LIN {X 0,Y 704.416,Z 634.552,A -85,B 0,C 180,E1 -3430.383,E2 -3430.383} C_VEL
LIN {X 0,Y 704.53,Z 624.148,A -85,B 0,C 180,E1 -3430.889,E2 -3430.889} C_VEL
LIN {X 0,Y 704.712,Z 613.331,A -85,B 0,C 180,E1 -3431.321,E2 -3431.321} C_VEL
LIN {X 0,Y 704.817,Z 602.117,A -85,B 0,C 180,E1 -3431.683,E2 -3431.683} C_VEL
LIN {X 0,Y 704.875,Z 590.492,A -85,B 0,C 180,E1 -3431.972,E2 -3431.972} C_VEL
LIN {X 0,Y 704.941,Z 578.231,A -85,B 0,C 180,E1 -3432.19,E2 -3432.19} C_VEL
LIN {X 0,Y 705.133,Z 516.872,A -85,B 0,C 180,E1 -3432.832,E2 -3432.832} C_VEL
LIN {X 0,Y 705.313,Z 446.172,A -85,B 0,C 180,E1 -3433.553,E2 -3433.553} C_VEL
LIN {X 0,Y 704.909,Z 442.652,A -85,B 0,C 180,E1 -3433.636,E2 -3433.636} C_VEL
LIN {X 0,Y 703.676,Z 438.808,A -85,B 0,C 180,E1 -3433.829,E2 -3433.829} C_VEL
LIN {X 0,Y 701.394,Z 434.303,A -85,B 0,C 180,E1 -3434.192,E2 -3434.192} C_VEL
LIN {X 0,Y 698.323,Z 427.937,A -85,B 0,C 180,E1 -3434.84,E2 -3434.84} C_VEL
LIN {X 0,Y 697.717,Z 423.757,A -85,B 0,C 180,E1 -3435.236,E2 -3435.236} C_VEL
LIN {X 0,Y 698.092,Z 392.579,A -85,B 0,C 180,E1 -3438.122,E2 -3438.122} C_VEL
LIN {X 0,Y 698.45,Z 360.795,A -85,B 0,C 180,E1 -3441.048,E2 -3441.048} C_VEL
LIN {X 0,Y 698.726,Z 332.913,A -85,B 0,C 180,E1 -3443.64,E2 -3443.64} C_VEL
LIN {X 0,Y 698.786,Z 319.402,A -85,B 0,C 180,E1 -3444.898,E2 -3444.898} C_VEL
LIN {X 0,Y 697.086,Z 311.216,A -85,B 0,C 180,E1 -3445.739,E2 -3445.739} C_VEL
LIN {X 0,Y 697.089,Z 311.207,A -85,B 0,C 180,E1 -3448.182,E2 -3448.182} C_VEL
LIN {X 0,Y 697.083,Z 311.208,A -85,B 0,C 180,E1 -3450.828,E2 -3450.828} C_VEL
LIN {X 0,Y 697.065,Z 311.215,A -85,B 0,C 180,E1 -3453.486,E2 -3453.486} C_VEL
LIN {X 0,Y 697.085,Z 311.208,A -85,B 0,C 180,E1 -3455.648,E2 -3455.648} C_VEL
LIN {X 0,Y 697.071,Z 311.207,A -85,B 0,C 180,E1 -3458.392,E2 -3458.392} C_VEL
LIN {X 0,Y 697.107,Z 311.212,A -85,B 0,C 180,E1 -3461.097,E2 -3461.097} C_VEL
LIN {X 0,Y 697.065,Z 311.208,A -85,B 0,C 180,E1 -3463.656,E2 -3463.656} C_VEL
LIN {X 0,Y 697.067,Z 311.207,A -85,B 0,C 180,E1 -3466.105,E2 -3466.105} C_VEL
LIN {X 0,Y 697.088,Z 311.21,A -85,B 0,C 180,E1 -3468.457,E2 -3468.457} C_VEL
LIN {X 0,Y 697.069,Z 311.218,A -85,B 0,C 180,E1 -3470.724,E2 -3470.724} C_VEL
LIN {X 0,Y 697.066,Z 311.207,A -85,B 0,C 180,E1 -3473.502,E2 -3473.502} C_VEL
LIN {X 0,Y 697.074,Z 311.207,A -85,B 0,C 180,E1 -3475.757,E2 -3475.757} C_VEL
LIN {X 0,Y 697.089,Z 311.214,A -85,B 0,C 180,E1 -3478.5,E2 -3478.5} C_VEL
LIN {X 0,Y 697.077,Z 311.206,A -85,B 0,C 180,E1 -3481.163,E2 -3481.163} C_VEL
LIN {X 0,Y 697.084,Z 311.205,A -85,B 0,C 180,E1 -3483.418,E2 -3483.418} C_VEL
LIN {X 0,Y 697.069,Z 311.218,A -85,B 0,C 180,E1 -3486.122,E2 -3486.122} C_VEL
LIN {X 0,Y 697.09,Z 311.205,A -85,B 0,C 180,E1 -3488.793,E2 -3488.793} C_VEL
LIN {X 0,Y 697.092,Z 311.205,A -85,B 0,C 180,E1 -3491.244,E2 -3491.244} C_VEL
LIN {X 0,Y 697.099,Z 311.211,A -85,B 0,C 180,E1 -3493.66,E2 -3493.66} C_VEL
LIN {X 0,Y 697.074,Z 311.213,A -85,B 0,C 180,E1 -3496.045,E2 -3496.045} C_VEL
LIN {X 0,Y 697.075,Z 311.216,A -85,B 0,C 180,E1 -3497.818,E2 -3497.818} C_VEL
LIN {X 0,Y 697.102,Z 311.206,A -85,B 0,C 180,E1 -3500.165,E2 -3500.165} C_VEL
LIN {X 0,Y 697.077,Z 311.215,A -85,B 0,C 180,E1 -3501.44,E2 -3501.44} C_VEL
LIN {X 0,Y 698.413,Z 316.046,A -85,B 0,C 180,E1 -3501.529,E2 -3501.529} C_VEL
LIN {X 0,Y 698.13,Z 433.864,A -85,B 0,C 180,E1 -3502.759,E2 -3502.759} C_VEL
LIN {X 0,Y 698.082,Z 445.644,A -85,B 0,C 180,E1 -3502.958,E2 -3502.958} C_VEL
LIN {X 0,Y 698.021,Z 457.462,A -85,B 0,C 180,E1 -3503.243,E2 -3503.243} C_VEL
LIN {X 0,Y 697.874,Z 469.115,A -85,B 0,C 180,E1 -3503.613,E2 -3503.613} C_VEL
LIN {X 0,Y 697.762,Z 478.918,A -85,B 0,C 180,E1 -3503.998,E2 -3503.998} C_VEL
LIN {X 0,Y 697.617,Z 489.914,A -85,B 0,C 180,E1 -3504.527,E2 -3504.527} C_VEL
LIN {X 0,Y 697.48,Z 499.897,A -85,B 0,C 180,E1 -3505.103,E2 -3505.103} C_VEL
LIN {X 0,Y 697.284,Z 510.292,A -85,B 0,C 180,E1 -3505.824,E2 -3505.824} C_VEL
LIN {X 0,Y 697.128,Z 519.035,A -85,B 0,C 180,E1 -3506.544,E2 -3506.544} C_VEL
LIN {X 0,Y 697.067,Z 526.496,A -85,B 0,C 180,E1 -3507.264,E2 -3507.264} C_VEL
LIN {X 0,Y 696.868,Z 534.07,A -85,B 0,C 180,E1 -3508.128,E2 -3508.128} C_VEL
LIN {X 0,Y 696.763,Z 539.463,A -85,B 0,C 180,E1 -3508.848,E2 -3508.848} C_VEL
LIN {X 0,Y 696.766,Z 544.86,A -85,B 0,C 180,E1 -3509.712,E2 -3509.712} C_VEL
LIN {X 0,Y 696.669,Z 549.315,A -85,B 0,C 180,E1 -3510.576,E2 -3510.576} C_VEL
LIN {X 0,Y 696.634,Z 553.802,A -85,B 0,C 180,E1 -3511.729,E2 -3511.729} C_VEL
LIN {X 0,Y 696.664,Z 556.881,A -85,B 0,C 180,E1 -3512.882,E2 -3512.882} C_VEL
LIN {X 0,Y 696.679,Z 558.012,A -85,B 0,C 180,E1 -3513.459,E2 -3513.459} C_VEL
LIN {X 0,Y 696.666,Z 559.13,A -85,B 0,C 180,E1 -3514.614,E2 -3514.614} C_VEL
LIN {X 0,Y 696.659,Z 558.934,A -85,B 0,C 180,E1 -3515.771,E2 -3515.771} C_VEL
LIN {X 0,Y 696.682,Z 557.437,A -85,B 0,C 180,E1 -3516.93,E2 -3516.93} C_VEL
LIN {X 0,Y 696.658,Z 556.281,A -85,B 0,C 180,E1 -3517.511,E2 -3517.511} C_VEL
LIN {X 0,Y 696.697,Z 552.763,A -85,B 0,C 180,E1 -3518.674,E2 -3518.674} C_VEL
LIN {X 0,Y 696.733,Z 547.682,A -85,B 0,C 180,E1 -3519.841,E2 -3519.841} C_VEL
LIN {X 0,Y 696.809,Z 542.835,A -85,B 0,C 180,E1 -3520.718,E2 -3520.718} C_VEL
LIN {X 0,Y 696.896,Z 536.913,A -85,B 0,C 180,E1 -3521.597,E2 -3521.597} C_VEL
LIN {X 0,Y 696.995,Z 529.74,A -85,B 0,C 180,E1 -3522.478,E2 -3522.478} C_VEL
LIN {X 0,Y 697.133,Z 522.817,A -85,B 0,C 180,E1 -3523.202,E2 -3523.202} C_VEL
LIN {X 0,Y 697.22,Z 514.383,A -85,B 0,C 180,E1 -3523.952,E2 -3523.952} C_VEL
LIN {X 0,Y 697.374,Z 504.458,A -85,B 0,C 180,E1 -3524.691,E2 -3524.691} C_VEL
LIN {X 0,Y 697.537,Z 493.912,A -85,B 0,C 180,E1 -3525.347,E2 -3525.347} C_VEL
LIN {X 0,Y 697.678,Z 483.686,A -85,B 0,C 180,E1 -3525.878,E2 -3525.878} C_VEL
LIN {X 0,Y 697.815,Z 472.333,A -85,B 0,C 180,E1 -3526.361,E2 -3526.361} C_VEL
LIN {X 0,Y 697.97,Z 460.217,A -85,B 0,C 180,E1 -3526.769,E2 -3526.769} C_VEL
LIN {X 0,Y 698.056,Z 448.742,A -85,B 0,C 180,E1 -3527.068,E2 -3527.068} C_VEL
LIN {X 0,Y 698.118,Z 436.727,A -85,B 0,C 180,E1 -3527.292,E2 -3527.292} C_VEL
LIN {X 0,Y 698.2,Z 406.687,A -85,B 0,C 180,E1 -3527.625,E2 -3527.625} C_VEL
LIN {X 0,Y 698.179,Z 314.933,A -85,B 0,C 180,E1 -3528.578,E2 -3528.578} C_VEL
LIN {X 0,Y 697.077,Z 311.216,A -85,B 0,C 180,E1 -3528.658,E2 -3528.658} C_VEL
LIN {X 0,Y 697.054,Z 311.212,A -85,B 0,C 180,E1 -3531.208,E2 -3531.208} C_VEL
LIN {X 0,Y 697.029,Z 311.217,A -85,B 0,C 180,E1 -3533.87,E2 -3533.87} C_VEL
LIN {X 0,Y 697.018,Z 311.223,A -85,B 0,C 180,E1 -3536.242,E2 -3536.242} C_VEL
LIN {X 0,Y 697.033,Z 311.22,A -85,B 0,C 180,E1 -3538.184,E2 -3538.184} C_VEL
LIN {X 0,Y 697.036,Z 311.213,A -85,B 0,C 180,E1 -3540.83,E2 -3540.83} C_VEL
LIN {X 0,Y 697.04,Z 311.212,A -85,B 0,C 180,E1 -3542.864,E2 -3542.864} C_VEL
LIN {X 0,Y 697.035,Z 311.213,A -85,B 0,C 180,E1 -3545.651,E2 -3545.651} C_VEL
LIN {X 0,Y 697.057,Z 311.216,A -85,B 0,C 180,E1 -3548.391,E2 -3548.391} C_VEL
LIN {X 0,Y 697.044,Z 311.21,A -85,B 0,C 180,E1 -3551.091,E2 -3551.091} C_VEL
LIN {X 0,Y 697.038,Z 311.219,A -85,B 0,C 180,E1 -3553.898,E2 -3553.898} C_VEL
LIN {X 0,Y 697.036,Z 311.217,A -85,B 0,C 180,E1 -3556.346,E2 -3556.346} C_VEL
LIN {X 0,Y 697.042,Z 311.209,A -85,B 0,C 180,E1 -3558.909,E2 -3558.909} C_VEL
LIN {X 0,Y 697.053,Z 311.212,A -85,B 0,C 180,E1 -3561.61,E2 -3561.61} C_VEL
LIN {X 0,Y 697.035,Z 311.211,A -85,B 0,C 180,E1 -3564.349,E2 -3564.349} C_VEL
LIN {X 0,Y 697.054,Z 311.208,A -85,B 0,C 180,E1 -3567.137,E2 -3567.137} C_VEL
LIN {X 0,Y 697.039,Z 311.21,A -85,B 0,C 180,E1 -3569.17,E2 -3569.17} C_VEL
LIN {X 0,Y 697.051,Z 311.209,A -85,B 0,C 180,E1 -3571.162,E2 -3571.162} C_VEL
LIN {X 0,Y 697.034,Z 311.215,A -85,B 0,C 180,E1 -3573.426,E2 -3573.426} C_VEL
LIN {X 0,Y 697.047,Z 311.219,A -85,B 0,C 180,E1 -3575.669,E2 -3575.669} C_VEL
LIN {X 0,Y 697.04,Z 311.211,A -85,B 0,C 180,E1 -3578.173,E2 -3578.173} C_VEL
LIN {X 0,Y 697.052,Z 311.21,A -85,B 0,C 180,E1 -3580.836,E2 -3580.836} C_VEL
LIN {X 0,Y 697.055,Z 311.213,A -85,B 0,C 180,E1 -3583.057,E2 -3583.057} C_VEL
LIN {X 0,Y 697.116,Z 311.212,A -85,B 0,C 180,E1 -3585.47,E2 -3585.47} C_VEL
LIN {X 0,Y 698.281,Z 315.996,A -85,B 0,C 180,E1 -3585.551,E2 -3585.551} C_VEL
LIN {X 0,Y 698.085,Z 434.452,A -85,B 0,C 180,E1 -3586.798,E2 -3586.798} C_VEL
LIN {X 0,Y 697.919,Z 448.239,A -85,B 0,C 180,E1 -3587.055,E2 -3587.055} C_VEL
LIN {X 0,Y 697.849,Z 460.688,A -85,B 0,C 180,E1 -3587.39,E2 -3587.39} C_VEL
LIN {X 0,Y 697.701,Z 471.338,A -85,B 0,C 180,E1 -3587.755,E2 -3587.755} C_VEL
LIN {X 0,Y 697.531,Z 483.202,A -85,B 0,C 180,E1 -3588.267,E2 -3588.267} C_VEL
LIN {X 0,Y 697.38,Z 493.02,A -85,B 0,C 180,E1 -3588.778,E2 -3588.778} C_VEL
LIN {X 0,Y 697.259,Z 503.504,A -85,B 0,C 180,E1 -3589.436,E2 -3589.436} C_VEL
LIN {X 0,Y 697.073,Z 512.639,A -85,B 0,C 180,E1 -3590.114,E2 -3590.114} C_VEL
LIN {X 0,Y 697.012,Z 519.975,A -85,B 0,C 180,E1 -3590.747,E2 -3590.747} C_VEL
LIN {X 0,Y 696.868,Z 528.488,A -85,B 0,C 180,E1 -3591.619,E2 -3591.619} C_VEL
LIN {X 0,Y 696.764,Z 535.677,A -85,B 0,C 180,E1 -3592.491,E2 -3592.491} C_VEL
LIN {X 0,Y 696.728,Z 541.669,A -85,B 0,C 180,E1 -3593.361,E2 -3593.361} C_VEL
LIN {X 0,Y 696.663,Z 546.618,A -85,B 0,C 180,E1 -3594.229,E2 -3594.229} C_VEL
LIN {X 0,Y 696.697,Z 550.636,A -85,B 0,C 180,E1 -3595.098,E2 -3595.098} C_VEL
LIN {X 0,Y 696.601,Z 553.765,A -85,B 0,C 180,E1 -3595.964,E2 -3595.964} C_VEL
LIN {X 0,Y 696.635,Z 556.64,A -85,B 0,C 180,E1 -3597.118,E2 -3597.118} C_VEL
LIN {X 0,Y 696.596,Z 558.138,A -85,B 0,C 180,E1 -3598.271,E2 -3598.271} C_VEL
LIN {X 0,Y 696.572,Z 558.438,A -85,B 0,C 180,E1 -3598.847,E2 -3598.847} C_VEL
LIN {X 0,Y 696.551,Z 558.045,A -85,B 0,C 180,E1 -3600,E2 -3600} C_VEL
LIN {X 0,Y 696.576,Z 556.29,A -85,B 0,C 180,E1 -3601.152,E2 -3601.152} C_VEL
LIN {X 0,Y 696.651,Z 553.124,A -85,B 0,C 180,E1 -3602.305,E2 -3602.305} C_VEL
LIN {X 0,Y 696.681,Z 549.882,A -85,B 0,C 180,E1 -3603.17,E2 -3603.17} C_VEL
LIN {X 0,Y 696.655,Z 545.754,A -85,B 0,C 180,E1 -3604.036,E2 -3604.036} C_VEL
LIN {X 0,Y 696.797,Z 539.655,A -85,B 0,C 180,E1 -3605.046,E2 -3605.046} C_VEL
LIN {X 0,Y 696.815,Z 533.283,A -85,B 0,C 180,E1 -3605.914,E2 -3605.914} C_VEL
LIN {X 0,Y 696.901,Z 525.644,A -85,B 0,C 180,E1 -3606.782,E2 -3606.782} C_VEL
LIN {X 0,Y 697.042,Z 518.237,A -85,B 0,C 180,E1 -3607.506,E2 -3607.506} C_VEL
LIN {X 0,Y 697.183,Z 508.476,A -85,B 0,C 180,E1 -3608.304,E2 -3608.304} C_VEL
LIN {X 0,Y 697.343,Z 498.984,A -85,B 0,C 180,E1 -3608.957,E2 -3608.957} C_VEL
LIN {X 0,Y 697.517,Z 488.951,A -85,B 0,C 180,E1 -3609.537,E2 -3609.537} C_VEL
LIN {X 0,Y 697.653,Z 478.255,A -85,B 0,C 180,E1 -3610.053,E2 -3610.053} C_VEL
LIN {X 0,Y 697.775,Z 466.28,A -85,B 0,C 180,E1 -3610.519,E2 -3610.519} C_VEL
LIN {X 0,Y 697.871,Z 454.325,A -85,B 0,C 180,E1 -3610.884,E2 -3610.884} C_VEL
LIN {X 0,Y 697.995,Z 440.597,A -85,B 0,C 180,E1 -3611.193,E2 -3611.193} C_VEL
LIN {X 0,Y 698.061,Z 426.048,A -85,B 0,C 180,E1 -3611.393,E2 -3611.393} C_VEL
LIN {X 0,Y 698.263,Z 315.137,A -85,B 0,C 180,E1 -3612.544,E2 -3612.544} C_VEL
LIN {X 0,Y 697.145,Z 311.208,A -85,B 0,C 180,E1 -3612.623,E2 -3612.623} C_VEL
LIN {X 0,Y 697.147,Z 311.199,A -85,B 0,C 180,E1 -3615.302,E2 -3615.302} C_VEL
LIN {X 0,Y 697.1,Z 311.214,A -85,B 0,C 180,E1 -3618.149,E2 -3618.149} C_VEL
LIN {X 0,Y 697.091,Z 311.209,A -85,B 0,C 180,E1 -3620.59,E2 -3620.59} C_VEL
LIN {X 0,Y 697.071,Z 311.208,A -85,B 0,C 180,E1 -3623.072,E2 -3623.072} C_VEL
LIN {X 0,Y 697.057,Z 311.214,A -85,B 0,C 180,E1 -3625.6,E2 -3625.6} C_VEL
LIN {X 0,Y 697.094,Z 311.209,A -85,B 0,C 180,E1 -3628.181,E2 -3628.181} C_VEL
LIN {X 0,Y 697.068,Z 311.207,A -85,B 0,C 180,E1 -3630.828,E2 -3630.828} C_VEL
LIN {X 0,Y 697.065,Z 311.217,A -85,B 0,C 180,E1 -3633.485,E2 -3633.485} C_VEL
LIN {X 0,Y 697.085,Z 311.213,A -85,B 0,C 180,E1 -3635.647,E2 -3635.647} C_VEL
LIN {X 0,Y 697.067,Z 311.206,A -85,B 0,C 180,E1 -3638.392,E2 -3638.392} C_VEL
LIN {X 0,Y 697.096,Z 311.21,A -85,B 0,C 180,E1 -3641.096,E2 -3641.096} C_VEL
LIN {X 0,Y 697.051,Z 311.209,A -85,B 0,C 180,E1 -3643.897,E2 -3643.897} C_VEL
LIN {X 0,Y 697.037,Z 311.211,A -85,B 0,C 180,E1 -3646.346,E2 -3646.346} C_VEL
LIN {X 0,Y 697.057,Z 311.214,A -85,B 0,C 180,E1 -3649.219,E2 -3649.219} C_VEL
LIN {X 0,Y 697.06,Z 311.209,A -85,B 0,C 180,E1 -3651.609,E2 -3651.609} C_VEL
LIN {X 0,Y 697.03,Z 311.217,A -85,B 0,C 180,E1 -3654.349,E2 -3654.349} C_VEL
LIN {X 0,Y 697.037,Z 311.214,A -85,B 0,C 180,E1 -3657.136,E2 -3657.136} C_VEL
LIN {X 0,Y 697.052,Z 311.211,A -85,B 0,C 180,E1 -3659.79,E2 -3659.79} C_VEL
LIN {X 0,Y 697.04,Z 311.221,A -85,B 0,C 180,E1 -3662.468,E2 -3662.468} C_VEL
LIN {X 0,Y 697.051,Z 311.256,A -85,B 0,C 180,E1 -3664.24,E2 -3664.24} C_VEL
LIN {X 0,Y 698.645,Z 320.018,A -85,B 0,C 180,E1 -3665.097,E2 -3665.097} C_VEL
LIN {X 0,Y 698.401,Z 349.089,A -85,B 0,C 180,E1 -3667.753,E2 -3667.753} C_VEL
LIN {X 0,Y 698.155,Z 376.319,A -85,B 0,C 180,E1 -3670.208,E2 -3670.208} C_VEL
LIN {X 0,Y 697.83,Z 403.417,A -85,B 0,C 180,E1 -3672.625,E2 -3672.625} C_VEL
LIN {X 0,Y 697.623,Z 432.113,A -85,B 0,C 180,E1 -3675.165,E2 -3675.165} C_VEL
LIN {X 0,Y 697.449,Z 444.539,A -85,B 0,C 180,E1 -3676.266,E2 -3676.266} C_VEL
LIN {X 0,Y 698.446,Z 452.348,A -85,B 0,C 180,E1 -3676.369,E2 -3676.369} C_VEL
LIN {X 0,Y 698.04,Z 582.997,A -85,B 0,C 180,E1 -3677.725,E2 -3677.725} C_VEL
LIN {X 0,Y 697.958,Z 597.77,A -85,B 0,C 180,E1 -3677.999,E2 -3677.999} C_VEL
LIN {X 0,Y 697.833,Z 610.65,A -85,B 0,C 180,E1 -3678.346,E2 -3678.346} C_VEL
LIN {X 0,Y 697.655,Z 623.019,A -85,B 0,C 180,E1 -3678.783,E2 -3678.783} C_VEL
LIN {X 0,Y 697.483,Z 635.95,A -85,B 0,C 180,E1 -3679.366,E2 -3679.366} C_VEL
LIN {X 0,Y 697.346,Z 647.324,A -85,B 0,C 180,E1 -3680,E2 -3680} C_VEL
LIN {X 0,Y 697.16,Z 658.402,A -85,B 0,C 180,E1 -3680.749,E2 -3680.749} C_VEL
LIN {X 0,Y 697.005,Z 669.021,A -85,B 0,C 180,E1 -3681.621,E2 -3681.621} C_VEL
LIN {X 0,Y 696.892,Z 677.791,A -85,B 0,C 180,E1 -3682.492,E2 -3682.492} C_VEL
LIN {X 0,Y 696.797,Z 686.202,A -85,B 0,C 180,E1 -3683.506,E2 -3683.506} C_VEL
LIN {X 0,Y 696.683,Z 693.878,A -85,B 0,C 180,E1 -3684.674,E2 -3684.674} C_VEL
LIN {X 0,Y 696.648,Z 699.022,A -85,B 0,C 180,E1 -3685.675,E2 -3685.675} C_VEL
LIN {X 0,Y 696.668,Z 702.489,A -85,B 0,C 180,E1 -3686.541,E2 -3686.541} C_VEL
LIN {X 0,Y 696.633,Z 705.854,A -85,B 0,C 180,E1 -3687.695,E2 -3687.695} C_VEL
LIN {X 0,Y 696.569,Z 707.841,A -85,B 0,C 180,E1 -3688.848,E2 -3688.848} C_VEL
LIN {X 0,Y 696.551,Z 708.5,A -85,B 0,C 180,E1 -3690,E2 -3690} C_VEL
LIN {X 0,Y 696.569,Z 707.84,A -85,B 0,C 180,E1 -3691.152,E2 -3691.152} C_VEL
LIN {X 0,Y 696.633,Z 705.852,A -85,B 0,C 180,E1 -3692.305,E2 -3692.305} C_VEL
LIN {X 0,Y 696.668,Z 702.487,A -85,B 0,C 180,E1 -3693.458,E2 -3693.458} C_VEL
LIN {X 0,Y 696.699,Z 697.646,A -85,B 0,C 180,E1 -3694.613,E2 -3694.613} C_VEL
LIN {X 0,Y 696.72,Z 691.176,A -85,B 0,C 180,E1 -3695.77,E2 -3695.77} C_VEL
LIN {X 0,Y 696.802,Z 683.979,A -85,B 0,C 180,E1 -3696.783,E2 -3696.783} C_VEL
LIN {X 0,Y 696.928,Z 675.084,A -85,B 0,C 180,E1 -3697.798,E2 -3697.798} C_VEL
LIN {X 0,Y 697.031,Z 665.75,A -85,B 0,C 180,E1 -3698.669,E2 -3698.669} C_VEL
LIN {X 0,Y 697.25,Z 654.358,A -85,B 0,C 180,E1 -3699.541,E2 -3699.541} C_VEL
LIN {X 0,Y 697.414,Z 642.364,A -85,B 0,C 180,E1 -3700.291,E2 -3700.291} C_VEL
LIN {X 0,Y 697.537,Z 629.856,A -85,B 0,C 180,E1 -3700.926,E2 -3700.926} C_VEL
LIN {X 0,Y 697.776,Z 616.228,A -85,B 0,C 180,E1 -3701.472,E2 -3701.472} C_VEL
LIN {X 0,Y 697.88,Z 603.07,A -85,B 0,C 180,E1 -3701.874,E2 -3701.874} C_VEL
LIN {X 0,Y 698.003,Z 588.739,A -85,B 0,C 180,E1 -3702.184,E2 -3702.184} C_VEL
LIN {X 0,Y 698.128,Z 573.562,A -85,B 0,C 180,E1 -3702.384,E2 -3702.384} C_VEL
LIN {X 0,Y 698.28,Z 450.581,A -85,B 0,C 180,E1 -3703.653,E2 -3703.653} C_VEL
LIN {X 0,Y 697.45,Z 444.438,A -85,B 0,C 180,E1 -3703.743,E2 -3703.743} C_VEL
LIN {X 0,Y 697.723,Z 418.64,A -85,B 0,C 180,E1 -3706.026,E2 -3706.026} C_VEL
LIN {X 0,Y 698.033,Z 388.214,A -85,B 0,C 180,E1 -3708.73,E2 -3708.73} C_VEL
LIN {X 0,Y 698.298,Z 361.073,A -85,B 0,C 180,E1 -3711.168,E2 -3711.168} C_VEL
LIN {X 0,Y 698.497,Z 335.496,A -85,B 0,C 180,E1 -3713.491,E2 -3713.491} C_VEL
LIN {X 0,Y 698.627,Z 320.105,A -85,B 0,C 180,E1 -3714.904,E2 -3714.904} C_VEL
LIN {X 0,Y 697.069,Z 311.217,A -85,B 0,C 180,E1 -3715.779,E2 -3715.779} C_VEL
LIN {X 0,Y 697.03,Z 311.216,A -85,B 0,C 180,E1 -3718.184,E2 -3718.184} C_VEL
LIN {X 0,Y 697.05,Z 311.211,A -85,B 0,C 180,E1 -3720.21,E2 -3720.21} C_VEL
LIN {X 0,Y 697.05,Z 311.209,A -85,B 0,C 180,E1 -3722.425,E2 -3722.425} C_VEL
LIN {X 0,Y 697.03,Z 311.215,A -85,B 0,C 180,E1 -3724.945,E2 -3724.945} C_VEL
LIN {X 0,Y 697.027,Z 311.221,A -85,B 0,C 180,E1 -3727.451,E2 -3727.451} C_VEL
LIN {X 0,Y 697.047,Z 311.21,A -85,B 0,C 180,E1 -3730.208,E2 -3730.208} C_VEL
LIN {X 0,Y 697.001,Z 311.22,A -85,B 0,C 180,E1 -3732.81,E2 -3732.81} C_VEL
LIN {X 0,Y 697.052,Z 311.218,A -85,B 0,C 180,E1 -3735.299,E2 -3735.299} C_VEL
LIN {X 0,Y 697.013,Z 311.214,A -85,B 0,C 180,E1 -3738.043,E2 -3738.043} C_VEL
LIN {X 0,Y 697.051,Z 311.209,A -85,B 0,C 180,E1 -3739.976,E2 -3739.976} C_VEL
LIN {X 0,Y 697.034,Z 311.216,A -85,B 0,C 180,E1 -3742.548,E2 -3742.548} C_VEL
LIN {X 0,Y 697.07,Z 311.215,A -85,B 0,C 180,E1 -3745.057,E2 -3745.057} C_VEL
LIN {X 0,Y 697.07,Z 311.21,A -85,B 0,C 180,E1 -3747.821,E2 -3747.821} C_VEL
LIN {X 0,Y 697.063,Z 311.22,A -85,B 0,C 180,E1 -3750.503,E2 -3750.503} C_VEL
LIN {X 0,Y 697.059,Z 311.214,A -85,B 0,C 180,E1 -3753.116,E2 -3753.116} C_VEL
LIN {X 0,Y 697.114,Z 311.307,A -85,B 0,C 180,E1 -3754.662,E2 -3754.662} C_VEL
LIN {X 0,Y 698.436,Z 319.322,A -85,B 0,C 180,E1 -3755.406,E2 -3755.406} C_VEL
LIN {X 0,Y 698.396,Z 345.702,A -85,B 0,C 180,E1 -3757.753,E2 -3757.753} C_VEL
LIN {X 0,Y 698.204,Z 369.482,A -85,B 0,C 180,E1 -3759.904,E2 -3759.904} C_VEL
LIN {X 0,Y 698.03,Z 393.207,A -85,B 0,C 180,E1 -3762.043,E2 -3762.043} C_VEL
LIN {X 0,Y 697.669,Z 423.864,A -85,B 0,C 180,E1 -3764.869,E2 -3764.869} C_VEL
LIN {X 0,Y 697.532,Z 439.974,A -85,B 0,C 180,E1 -3766.32,E2 -3766.32} C_VEL
LIN {X 0,Y 698.391,Z 447.928,A -85,B 0,C 180,E1 -3766.419,E2 -3766.419} C_VEL
LIN {X 0,Y 698.081,Z 577.12,A -85,B 0,C 180,E1 -3767.763,E2 -3767.763} C_VEL
LIN {X 0,Y 697.985,Z 589.7,A -85,B 0,C 180,E1 -3767.981,E2 -3767.981} C_VEL
LIN {X 0,Y 697.839,Z 601.509,A -85,B 0,C 180,E1 -3768.273,E2 -3768.273} C_VEL
LIN {X 0,Y 697.724,Z 611.828,A -85,B 0,C 180,E1 -3768.601,E2 -3768.601} C_VEL
LIN {X 0,Y 697.551,Z 622.078,A -85,B 0,C 180,E1 -3769.001,E2 -3769.001} C_VEL
LIN {X 0,Y 697.425,Z 632.817,A -85,B 0,C 180,E1 -3769.512,E2 -3769.512} C_VEL
LIN {X 0,Y 697.308,Z 642.888,A -85,B 0,C 180,E1 -3770.085,E2 -3770.085} C_VEL
LIN {X 0,Y 697.185,Z 652.755,A -85,B 0,C 180,E1 -3770.75,E2 -3770.75} C_VEL
LIN {X 0,Y 697.023,Z 663.56,A -85,B 0,C 180,E1 -3771.622,E2 -3771.622} C_VEL
LIN {X 0,Y 696.896,Z 672.354,A -85,B 0,C 180,E1 -3772.492,E2 -3772.492} C_VEL
LIN {X 0,Y 696.786,Z 679.7,A -85,B 0,C 180,E1 -3773.362,E2 -3773.362} C_VEL
LIN {X 0,Y 696.721,Z 685.834,A -85,B 0,C 180,E1 -3774.23,E2 -3774.23} C_VEL
LIN {X 0,Y 696.725,Z 690.907,A -85,B 0,C 180,E1 -3775.098,E2 -3775.098} C_VEL
LIN {X 0,Y 696.633,Z 695.019,A -85,B 0,C 180,E1 -3775.964,E2 -3775.964} C_VEL
LIN {X 0,Y 696.669,Z 697.337,A -85,B 0,C 180,E1 -3776.542,E2 -3776.542} C_VEL
LIN {X 0,Y 696.634,Z 700.722,A -85,B 0,C 180,E1 -3777.695,E2 -3777.695} C_VEL
LIN {X 0,Y 696.574,Z 702.769,A -85,B 0,C 180,E1 -3778.848,E2 -3778.848} C_VEL
LIN {X 0,Y 696.55,Z 703.494,A -85,B 0,C 180,E1 -3780,E2 -3780} C_VEL
LIN {X 0,Y 696.572,Z 702.859,A -85,B 0,C 180,E1 -3781.153,E2 -3781.153} C_VEL
LIN {X 0,Y 696.633,Z 700.934,A -85,B 0,C 180,E1 -3782.305,E2 -3782.305} C_VEL
LIN {X 0,Y 696.669,Z 697.625,A -85,B 0,C 180,E1 -3783.459,E2 -3783.459} C_VEL
LIN {X 0,Y 696.7,Z 692.884,A -85,B 0,C 180,E1 -3784.613,E2 -3784.613} C_VEL
LIN {X 0,Y 696.705,Z 687.827,A -85,B 0,C 180,E1 -3785.547,E2 -3785.547} C_VEL
LIN {X 0,Y 696.798,Z 681.478,A -85,B 0,C 180,E1 -3786.494,E2 -3786.494} C_VEL
LIN {X 0,Y 696.857,Z 674.445,A -85,B 0,C 180,E1 -3787.363,E2 -3787.363} C_VEL
LIN {X 0,Y 696.957,Z 667.529,A -85,B 0,C 180,E1 -3788.089,E2 -3788.089} C_VEL
LIN {X 0,Y 697.065,Z 659.448,A -85,B 0,C 180,E1 -3788.815,E2 -3788.815} C_VEL
LIN {X 0,Y 697.228,Z 649.929,A -85,B 0,C 180,E1 -3789.542,E2 -3789.542} C_VEL
LIN {X 0,Y 697.38,Z 638.441,A -85,B 0,C 180,E1 -3790.277,E2 -3790.277} C_VEL
LIN {X 0,Y 697.538,Z 625.787,A -85,B 0,C 180,E1 -3790.926,E2 -3790.926} C_VEL
LIN {X 0,Y 697.734,Z 614.312,A -85,B 0,C 180,E1 -3791.399,E2 -3791.399} C_VEL
LIN {X 0,Y 697.827,Z 603.347,A -85,B 0,C 180,E1 -3791.765,E2 -3791.765} C_VEL
LIN {X 0,Y 697.927,Z 592.099,A -85,B 0,C 180,E1 -3792.057,E2 -3792.057} C_VEL
LIN {X 0,Y 698.021,Z 581.719,A -85,B 0,C 180,E1 -3792.257,E2 -3792.257} C_VEL
LIN {X 0,Y 698.113,Z 567.551,A -85,B 0,C 180,E1 -3792.439,E2 -3792.439} C_VEL
LIN {X 0,Y 698.389,Z 446.33,A -85,B 0,C 180,E1 -3793.688,E2 -3793.688} C_VEL
LIN {X 0,Y 697.497,Z 439.68,A -85,B 0,C 180,E1 -3793.775,E2 -3793.775} C_VEL
LIN {X 0,Y 697.717,Z 423.757,A -85,B 0,C 180,E1 -3795.236,E2 -3795.236} C_VEL
LIN {X 0,Y 697.138,Z 419.925,A -85,B 0,C 180,E1 -3795.602,E2 -3795.602} C_VEL
LIN {X 0,Y 691.543,Z 408.04,A -85,B 0,C 180,E1 -3796.832,E2 -3796.832} C_VEL
LIN {X 0,Y 690.973,Z 404.22,A -85,B 0,C 180,E1 -3797.204,E2 -3797.204} C_VEL
LIN {X 0,Y 691.299,Z 377.64,A -85,B 0,C 180,E1 -3799.673,E2 -3799.673} C_VEL
LIN {X 0,Y 691.587,Z 352.552,A -85,B 0,C 180,E1 -3802.008,E2 -3802.008} C_VEL
LIN {X 0,Y 691.897,Z 328.704,A -85,B 0,C 180,E1 -3804.242,E2 -3804.242} C_VEL
LIN {X 0,Y 691.863,Z 320.646,A -85,B 0,C 180,E1 -3805.004,E2 -3805.004} C_VEL
LIN {X 0,Y 690.042,Z 312.092,A -85,B 0,C 180,E1 -3805.88,E2 -3805.88} C_VEL
LIN {X 0,Y 690.041,Z 312.084,A -85,B 0,C 180,E1 -3808.496,E2 -3808.496} C_VEL
LIN {X 0,Y 690.041,Z 312.091,A -85,B 0,C 180,E1 -3811.178,E2 -3811.178} C_VEL
LIN {X 0,Y 690.039,Z 312.087,A -85,B 0,C 180,E1 -3813.657,E2 -3813.657} C_VEL
LIN {X 0,Y 690.032,Z 312.083,A -85,B 0,C 180,E1 -3816.069,E2 -3816.069} C_VEL
LIN {X 0,Y 690.047,Z 312.084,A -85,B 0,C 180,E1 -3818.592,E2 -3818.592} C_VEL
LIN {X 0,Y 690.065,Z 312.085,A -85,B 0,C 180,E1 -3821.311,E2 -3821.311} C_VEL
LIN {X 0,Y 690.043,Z 312.082,A -85,B 0,C 180,E1 -3823.887,E2 -3823.887} C_VEL
LIN {X 0,Y 690.035,Z 312.086,A -85,B 0,C 180,E1 -3826.349,E2 -3826.349} C_VEL
LIN {X 0,Y 690.052,Z 312.091,A -85,B 0,C 180,E1 -3828.716,E2 -3828.716} C_VEL
LIN {X 0,Y 690.049,Z 312.082,A -85,B 0,C 180,E1 -3831.408,E2 -3831.408} C_VEL
LIN {X 0,Y 690.037,Z 312.089,A -85,B 0,C 180,E1 -3834.299,E2 -3834.299} C_VEL
LIN {X 0,Y 690.02,Z 312.091,A -85,B 0,C 180,E1 -3836.759,E2 -3836.759} C_VEL
LIN {X 0,Y 690.036,Z 312.087,A -85,B 0,C 180,E1 -3838.822,E2 -3838.822} C_VEL
LIN {X 0,Y 690.044,Z 312.082,A -85,B 0,C 180,E1 -3841.505,E2 -3841.505} C_VEL
LIN {X 0,Y 690.009,Z 312.096,A -85,B 0,C 180,E1 -3844.119,E2 -3844.119} C_VEL
LIN {X 0,Y 690.042,Z 312.084,A -85,B 0,C 180,E1 -3846.679,E2 -3846.679} C_VEL
LIN {X 0,Y 690.055,Z 312.081,A -85,B 0,C 180,E1 -3849.19,E2 -3849.19} C_VEL
LIN {X 0,Y 690.05,Z 312.088,A -85,B 0,C 180,E1 -3851.659,E2 -3851.659} C_VEL
LIN {X 0,Y 690.036,Z 312.09,A -85,B 0,C 180,E1 -3854.093,E2 -3854.093} C_VEL
LIN {X 0,Y 690.092,Z 312.078,A -85,B 0,C 180,E1 -3857.097,E2 -3857.097} C_VEL
LIN {X 0,Y 690.09,Z 312.081,A -85,B 0,C 180,E1 -3860.064,E2 -3860.064} C_VEL
LIN {X 0,Y 690.036,Z 312.09,A -85,B 0,C 180,E1 -3861.297,E2 -3861.297} C_VEL
LIN {X 0,Y 691.437,Z 316.696,A -85,B 0,C 180,E1 -3861.389,E2 -3861.389} C_VEL
LIN {X 0,Y 691.226,Z 435.797,A -85,B 0,C 180,E1 -3862.65,E2 -3862.65} C_VEL
LIN {X 0,Y 691.172,Z 448.873,A -85,B 0,C 180,E1 -3862.887,E2 -3862.887} C_VEL
LIN {X 0,Y 691.043,Z 461.433,A -85,B 0,C 180,E1 -3863.215,E2 -3863.215} C_VEL
LIN {X 0,Y 690.924,Z 474.328,A -85,B 0,C 180,E1 -3863.663,E2 -3863.663} C_VEL
LIN {X 0,Y 690.75,Z 487.537,A -85,B 0,C 180,E1 -3864.253,E2 -3864.253} C_VEL
LIN {X 0,Y 690.554,Z 500.341,A -85,B 0,C 180,E1 -3864.981,E2 -3864.981} C_VEL
LIN {X 0,Y 690.352,Z 509.853,A -85,B 0,C 180,E1 -3865.636,E2 -3865.636} C_VEL
LIN {X 0,Y 690.209,Z 518.78,A -85,B 0,C 180,E1 -3866.364,E2 -3866.364} C_VEL
LIN {X 0,Y 690.073,Z 527.744,A -85,B 0,C 180,E1 -3867.237,E2 -3867.237} C_VEL
LIN {X 0,Y 689.873,Z 535.241,A -85,B 0,C 180,E1 -3868.109,E2 -3868.109} C_VEL
LIN {X 0,Y 689.749,Z 540.568,A -85,B 0,C 180,E1 -3868.836,E2 -3868.836} C_VEL
LIN {X 0,Y 689.746,Z 545.9,A -85,B 0,C 180,E1 -3869.709,E2 -3869.709} C_VEL
LIN {X 0,Y 689.654,Z 550.301,A -85,B 0,C 180,E1 -3870.582,E2 -3870.582} C_VEL
LIN {X 0,Y 689.586,Z 554.73,A -85,B 0,C 180,E1 -3871.746,E2 -3871.746} C_VEL
LIN {X 0,Y 689.627,Z 556.46,A -85,B 0,C 180,E1 -3872.329,E2 -3872.329} C_VEL
LIN {X 0,Y 689.632,Z 558.851,A -85,B 0,C 180,E1 -3873.494,E2 -3873.494} C_VEL
LIN {X 0,Y 689.607,Z 559.91,A -85,B 0,C 180,E1 -3874.661,E2 -3874.661} C_VEL
LIN {X 0,Y 689.622,Z 559.664,A -85,B 0,C 180,E1 -3875.83,E2 -3875.83} C_VEL
LIN {X 0,Y 689.636,Z 559.092,A -85,B 0,C 180,E1 -3876.415,E2 -3876.415} C_VEL
LIN {X 0,Y 689.63,Z 556.919,A -85,B 0,C 180,E1 -3877.588,E2 -3877.588} C_VEL
LIN {X 0,Y 689.661,Z 553.339,A -85,B 0,C 180,E1 -3878.763,E2 -3878.763} C_VEL
LIN {X 0,Y 689.74,Z 548.196,A -85,B 0,C 180,E1 -3879.941,E2 -3879.941} C_VEL
LIN {X 0,Y 689.791,Z 543.29,A -85,B 0,C 180,E1 -3880.828,E2 -3880.828} C_VEL
LIN {X 0,Y 689.898,Z 537.298,A -85,B 0,C 180,E1 -3881.716,E2 -3881.716} C_VEL
LIN {X 0,Y 690.03,Z 530.045,A -85,B 0,C 180,E1 -3882.606,E2 -3882.606} C_VEL
LIN {X 0,Y 690.148,Z 522.903,A -85,B 0,C 180,E1 -3883.35,E2 -3883.35} C_VEL
LIN {X 0,Y 690.273,Z 514.498,A -85,B 0,C 180,E1 -3884.096,E2 -3884.096} C_VEL
LIN {X 0,Y 690.437,Z 504.452,A -85,B 0,C 180,E1 -3884.842,E2 -3884.842} C_VEL
LIN {X 0,Y 690.603,Z 493.502,A -85,B 0,C 180,E1 -3885.519,E2 -3885.519} C_VEL
LIN {X 0,Y 690.788,Z 483.329,A -85,B 0,C 180,E1 -3886.04,E2 -3886.04} C_VEL
LIN {X 0,Y 690.935,Z 471.699,A -85,B 0,C 180,E1 -3886.528,E2 -3886.528} C_VEL
LIN {X 0,Y 691.072,Z 460.48,A -85,B 0,C 180,E1 -3886.904,E2 -3886.904} C_VEL
LIN {X 0,Y 691.143,Z 448.101,A -85,B 0,C 180,E1 -3887.221,E2 -3887.221} C_VEL
LIN {X 0,Y 691.215,Z 435.779,A -85,B 0,C 180,E1 -3887.442,E2 -3887.442} C_VEL
LIN {X 0,Y 691.462,Z 317.625,A -85,B 0,C 180,E1 -3888.691,E2 -3888.691} C_VEL
LIN {X 0,Y 690.049,Z 312.091,A -85,B 0,C 180,E1 -3888.785,E2 -3888.785} C_VEL
LIN {X 0,Y 690.001,Z 312.09,A -85,B 0,C 180,E1 -3891.435,E2 -3891.435} C_VEL
LIN {X 0,Y 690.006,Z 312.093,A -85,B 0,C 180,E1 -3893.989,E2 -3893.989} C_VEL
LIN {X 0,Y 689.981,Z 312.094,A -85,B 0,C 180,E1 -3895.882,E2 -3895.882} C_VEL
LIN {X 0,Y 689.988,Z 312.099,A -85,B 0,C 180,E1 -3898.498,E2 -3898.498} C_VEL
LIN {X 0,Y 689.997,Z 312.096,A -85,B 0,C 180,E1 -3900.502,E2 -3900.502} C_VEL
LIN {X 0,Y 690.003,Z 312.093,A -85,B 0,C 180,E1 -3902.588,E2 -3902.588} C_VEL
LIN {X 0,Y 690.011,Z 312.086,A -85,B 0,C 180,E1 -3905.354,E2 -3905.354} C_VEL
LIN {X 0,Y 690.001,Z 312.089,A -85,B 0,C 180,E1 -3907.645,E2 -3907.645} C_VEL
LIN {X 0,Y 690.016,Z 312.092,A -85,B 0,C 180,E1 -3910.418,E2 -3910.418} C_VEL
LIN {X 0,Y 689.978,Z 312.09,A -85,B 0,C 180,E1 -3913.036,E2 -3913.036} C_VEL
LIN {X 0,Y 690.04,Z 312.084,A -85,B 0,C 180,E1 -3915.54,E2 -3915.54} C_VEL
LIN {X 0,Y 689.973,Z 312.1,A -85,B 0,C 180,E1 -3917.931,E2 -3917.931} C_VEL
LIN {X 0,Y 689.986,Z 312.09,A -85,B 0,C 180,E1 -3920.491,E2 -3920.491} C_VEL
LIN {X 0,Y 689.997,Z 312.083,A -85,B 0,C 180,E1 -3922.476,E2 -3922.476} C_VEL
LIN {X 0,Y 690.012,Z 312.083,A -85,B 0,C 180,E1 -3924.646,E2 -3924.646} C_VEL
LIN {X 0,Y 690.048,Z 312.084,A -85,B 0,C 180,E1 -3927.453,E2 -3927.453} C_VEL
LIN {X 0,Y 690.01,Z 312.09,A -85,B 0,C 180,E1 -3930.171,E2 -3930.171} C_VEL
LIN {X 0,Y 689.987,Z 312.088,A -85,B 0,C 180,E1 -3932.818,E2 -3932.818} C_VEL
LIN {X 0,Y 690.006,Z 312.09,A -85,B 0,C 180,E1 -3935.405,E2 -3935.405} C_VEL
LIN {X 0,Y 689.984,Z 312.094,A -85,B 0,C 180,E1 -3937.938,E2 -3937.938} C_VEL
LIN {X 0,Y 689.993,Z 312.09,A -85,B 0,C 180,E1 -3940.427,E2 -3940.427} C_VEL
LIN {X 0,Y 690.028,Z 312.087,A -85,B 0,C 180,E1 -3942.88,E2 -3942.88} C_VEL
LIN {X 0,Y 690.049,Z 312.091,A -85,B 0,C 180,E1 -3945.337,E2 -3945.337} C_VEL
LIN {X 0,Y 691.401,Z 317.217,A -85,B 0,C 180,E1 -3945.426,E2 -3945.426} C_VEL
LIN {X 0,Y 691.144,Z 434.963,A -85,B 0,C 180,E1 -3946.685,E2 -3946.685} C_VEL
LIN {X 0,Y 690.98,Z 449.204,A -85,B 0,C 180,E1 -3946.954,E2 -3946.954} C_VEL
LIN {X 0,Y 690.877,Z 461.782,A -85,B 0,C 180,E1 -3947.298,E2 -3947.298} C_VEL
LIN {X 0,Y 690.713,Z 473.248,A -85,B 0,C 180,E1 -3947.704,E2 -3947.704} C_VEL
LIN {X 0,Y 690.563,Z 484.897,A -85,B 0,C 180,E1 -3948.221,E2 -3948.221} C_VEL
LIN {X 0,Y 690.401,Z 494.561,A -85,B 0,C 180,E1 -3948.738,E2 -3948.738} C_VEL
LIN {X 0,Y 690.296,Z 503.898,A -85,B 0,C 180,E1 -3949.328,E2 -3949.328} C_VEL
LIN {X 0,Y 690.091,Z 513.686,A -85,B 0,C 180,E1 -3950.064,E2 -3950.064} C_VEL
LIN {X 0,Y 689.975,Z 521.956,A -85,B 0,C 180,E1 -3950.799,E2 -3950.799} C_VEL
LIN {X 0,Y 689.845,Z 529.031,A -85,B 0,C 180,E1 -3951.534,E2 -3951.534} C_VEL
LIN {X 0,Y 689.742,Z 536.155,A -85,B 0,C 180,E1 -3952.414,E2 -3952.414} C_VEL
LIN {X 0,Y 689.674,Z 542.081,A -85,B 0,C 180,E1 -3953.293,E2 -3953.293} C_VEL
LIN {X 0,Y 689.61,Z 546.967,A -85,B 0,C 180,E1 -3954.17,E2 -3954.17} C_VEL
LIN {X 0,Y 689.631,Z 550.927,A -85,B 0,C 180,E1 -3955.047,E2 -3955.047} C_VEL
LIN {X 0,Y 689.52,Z 554.011,A -85,B 0,C 180,E1 -3955.922,E2 -3955.922} C_VEL
LIN {X 0,Y 689.557,Z 556.851,A -85,B 0,C 180,E1 -3957.089,E2 -3957.089} C_VEL
LIN {X 0,Y 689.522,Z 558.332,A -85,B 0,C 180,E1 -3958.253,E2 -3958.253} C_VEL
LIN {X 0,Y 689.468,Z 558.547,A -85,B 0,C 180,E1 -3959.418,E2 -3959.418} C_VEL
LIN {X 0,Y 689.462,Z 558.265,A -85,B 0,C 180,E1 -3960,E2 -3960} C_VEL
LIN {X 0,Y 689.494,Z 556.561,A -85,B 0,C 180,E1 -3961.164,E2 -3961.164} C_VEL
LIN {X 0,Y 689.59,Z 553.466,A -85,B 0,C 180,E1 -3962.328,E2 -3962.328} C_VEL
LIN {X 0,Y 689.602,Z 550.299,A -85,B 0,C 180,E1 -3963.202,E2 -3963.202} C_VEL
LIN {X 0,Y 689.602,Z 546.252,A -85,B 0,C 180,E1 -3964.077,E2 -3964.077} C_VEL
LIN {X 0,Y 689.744,Z 541.231,A -85,B 0,C 180,E1 -3964.952,E2 -3964.952} C_VEL
LIN {X 0,Y 689.797,Z 534.006,A -85,B 0,C 180,E1 -3965.974,E2 -3965.974} C_VEL
LIN {X 0,Y 689.915,Z 526.447,A -85,B 0,C 180,E1 -3966.851,E2 -3966.851} C_VEL
LIN {X 0,Y 690.052,Z 517.315,A -85,B 0,C 180,E1 -3967.729,E2 -3967.729} C_VEL
LIN {X 0,Y 690.22,Z 508.234,A -85,B 0,C 180,E1 -3968.462,E2 -3968.462} C_VEL
LIN {X 0,Y 690.364,Z 498.529,A -85,B 0,C 180,E1 -3969.122,E2 -3969.122} C_VEL
LIN {X 0,Y 690.583,Z 488.22,A -85,B 0,C 180,E1 -3969.708,E2 -3969.708} C_VEL
LIN {X 0,Y 690.715,Z 478.08,A -85,B 0,C 180,E1 -3970.191,E2 -3970.191} C_VEL
LIN {X 0,Y 690.833,Z 466.927,A -85,B 0,C 180,E1 -3970.626,E2 -3970.626} C_VEL
LIN {X 0,Y 690.945,Z 454.185,A -85,B 0,C 180,E1 -3971.013,E2 -3971.013} C_VEL
LIN {X 0,Y 691.055,Z 440.972,A -85,B 0,C 180,E1 -3971.307,E2 -3971.307} C_VEL
LIN {X 0,Y 691.117,Z 426.056,A -85,B 0,C 180,E1 -3971.509,E2 -3971.509} C_VEL
LIN {X 0,Y 691.36,Z 316.399,A -85,B 0,C 180,E1 -3972.668,E2 -3972.668} C_VEL
LIN {X 0,Y 690.097,Z 312.085,A -85,B 0,C 180,E1 -3972.754,E2 -3972.754} C_VEL
LIN {X 0,Y 690.1,Z 312.08,A -85,B 0,C 180,E1 -3975.905,E2 -3975.905} C_VEL
LIN {X 0,Y 690.051,Z 312.092,A -85,B 0,C 180,E1 -3978.341,E2 -3978.341} C_VEL
LIN {X 0,Y 690.044,Z 312.084,A -85,B 0,C 180,E1 -3980.953,E2 -3980.953} C_VEL
LIN {X 0,Y 690.047,Z 312.084,A -85,B 0,C 180,E1 -3983.321,E2 -3983.321} C_VEL
LIN {X 0,Y 690.011,Z 312.098,A -85,B 0,C 180,E1 -3985.881,E2 -3985.881} C_VEL
LIN {X 0,Y 690.048,Z 312.083,A -85,B 0,C 180,E1 -3988.495,E2 -3988.495} C_VEL
LIN {X 0,Y 690.035,Z 312.086,A -85,B 0,C 180,E1 -3991.178,E2 -3991.178} C_VEL
LIN {X 0,Y 690.039,Z 312.092,A -85,B 0,C 180,E1 -3993.657,E2 -3993.657} C_VEL
LIN {X 0,Y 690.032,Z 312.085,A -85,B 0,C 180,E1 -3996.068,E2 -3996.068} C_VEL
LIN {X 0,Y 690.043,Z 312.081,A -85,B 0,C 180,E1 -3998.592,E2 -3998.592} C_VEL
LIN {X 0,Y 690.031,Z 312.093,A -85,B 0,C 180,E1 -4001.308,E2 -4001.308} C_VEL
LIN {X 0,Y 690.028,Z 312.083,A -85,B 0,C 180,E1 -4003.886,E2 -4003.886} C_VEL
LIN {X 0,Y 690.009,Z 312.086,A -85,B 0,C 180,E1 -4006.347,E2 -4006.347} C_VEL
LIN {X 0,Y 689.992,Z 312.095,A -85,B 0,C 180,E1 -4008.711,E2 -4008.711} C_VEL
LIN {X 0,Y 690.035,Z 312.085,A -85,B 0,C 180,E1 -4011.409,E2 -4011.409} C_VEL
LIN {X 0,Y 689.981,Z 312.094,A -85,B 0,C 180,E1 -4014.305,E2 -4014.305} C_VEL
LIN {X 0,Y 689.996,Z 312.097,A -85,B 0,C 180,E1 -4016.758,E2 -4016.758} C_VEL
LIN {X 0,Y 690.002,Z 312.094,A -85,B 0,C 180,E1 -4018.82,E2 -4018.82} C_VEL
LIN {X 0,Y 690.014,Z 312.092,A -85,B 0,C 180,E1 -4020.839,E2 -4020.839} C_VEL
LIN {X 0,Y 689.996,Z 312.092,A -85,B 0,C 180,E1 -4023.294,E2 -4023.294} C_VEL
LIN {X 0,Y 690.017,Z 312.189,A -85,B 0,C 180,E1 -4024.119,E2 -4024.119} C_VEL
LIN {X 0,Y 691.685,Z 320.939,A -85,B 0,C 180,E1 -4024.989,E2 -4024.989} C_VEL
LIN {X 0,Y 691.461,Z 348.3,A -85,B 0,C 180,E1 -4027.517,E2 -4027.517} C_VEL
LIN {X 0,Y 691.165,Z 377.23,A -85,B 0,C 180,E1 -4030.154,E2 -4030.154} C_VEL
LIN {X 0,Y 690.8,Z 404.721,A -85,B 0,C 180,E1 -4032.632,E2 -4032.632} C_VEL
LIN {X 0,Y 690.571,Z 433.009,A -85,B 0,C 180,E1 -4035.16,E2 -4035.16} C_VEL
LIN {X 0,Y 690.429,Z 443.724,A -85,B 0,C 180,E1 -4036.114,E2 -4036.114} C_VEL
LIN {X 0,Y 691.519,Z 453.439,A -85,B 0,C 180,E1 -4036.248,E2 -4036.248} C_VEL
LIN {X 0,Y 691.097,Z 582.704,A -85,B 0,C 180,E1 -4037.6,E2 -4037.6} C_VEL
LIN {X 0,Y 690.99,Z 597.562,A -85,B 0,C 180,E1 -4037.876,E2 -4037.876} C_VEL
LIN {X 0,Y 690.841,Z 611.671,A -85,B 0,C 180,E1 -4038.263,E2 -4038.263} C_VEL
LIN {X 0,Y 690.653,Z 624.768,A -85,B 0,C 180,E1 -4038.742,E2 -4038.742} C_VEL
LIN {X 0,Y 690.465,Z 637.369,A -85,B 0,C 180,E1 -4039.331,E2 -4039.331} C_VEL
LIN {X 0,Y 690.335,Z 648.193,A -85,B 0,C 180,E1 -4039.953,E2 -4039.953} C_VEL
LIN {X 0,Y 690.138,Z 658.401,A -85,B 0,C 180,E1 -4040.654,E2 -4040.654} C_VEL
LIN {X 0,Y 689.941,Z 669.021,A -85,B 0,C 180,E1 -4041.535,E2 -4041.535} C_VEL
LIN {X 0,Y 689.841,Z 677.79,A -85,B 0,C 180,E1 -4042.415,E2 -4042.415} C_VEL
LIN {X 0,Y 689.721,Z 686.202,A -85,B 0,C 180,E1 -4043.44,E2 -4043.44} C_VEL
LIN {X 0,Y 689.635,Z 693.075,A -85,B 0,C 180,E1 -4044.479,E2 -4044.479} C_VEL
LIN {X 0,Y 689.612,Z 697.643,A -85,B 0,C 180,E1 -4045.339,E2 -4045.339} C_VEL
LIN {X 0,Y 689.569,Z 702.489,A -85,B 0,C 180,E1 -4046.506,E2 -4046.506} C_VEL
LIN {X 0,Y 689.542,Z 705.855,A -85,B 0,C 180,E1 -4047.671,E2 -4047.671} C_VEL
LIN {X 0,Y 689.487,Z 707.841,A -85,B 0,C 180,E1 -4048.836,E2 -4048.836} C_VEL
LIN {X 0,Y 689.462,Z 708.5,A -85,B 0,C 180,E1 -4050,E2 -4050} C_VEL
LIN {X 0,Y 689.487,Z 707.84,A -85,B 0,C 180,E1 -4051.164,E2 -4051.164} C_VEL
LIN {X 0,Y 689.542,Z 705.852,A -85,B 0,C 180,E1 -4052.329,E2 -4052.329} C_VEL
LIN {X 0,Y 689.569,Z 702.487,A -85,B 0,C 180,E1 -4053.494,E2 -4053.494} C_VEL
LIN {X 0,Y 689.612,Z 697.646,A -85,B 0,C 180,E1 -4054.661,E2 -4054.661} C_VEL
LIN {X 0,Y 689.66,Z 691.176,A -85,B 0,C 180,E1 -4055.829,E2 -4055.829} C_VEL
LIN {X 0,Y 689.743,Z 683.979,A -85,B 0,C 180,E1 -4056.853,E2 -4056.853} C_VEL
LIN {X 0,Y 689.861,Z 675.084,A -85,B 0,C 180,E1 -4057.878,E2 -4057.878} C_VEL
LIN {X 0,Y 689.998,Z 665.75,A -85,B 0,C 180,E1 -4058.758,E2 -4058.758} C_VEL
LIN {X 0,Y 690.23,Z 654.357,A -85,B 0,C 180,E1 -4059.639,E2 -4059.639} C_VEL
LIN {X 0,Y 690.398,Z 642.481,A -85,B 0,C 180,E1 -4060.39,E2 -4060.39} C_VEL
LIN {X 0,Y 690.545,Z 629.854,A -85,B 0,C 180,E1 -4061.038,E2 -4061.038} C_VEL
LIN {X 0,Y 690.81,Z 616.166,A -85,B 0,C 180,E1 -4061.589,E2 -4061.589} C_VEL
LIN {X 0,Y 690.943,Z 602.9,A -85,B 0,C 180,E1 -4061.995,E2 -4061.995} C_VEL
LIN {X 0,Y 691.06,Z 588.478,A -85,B 0,C 180,E1 -4062.308,E2 -4062.308} C_VEL
LIN {X 0,Y 691.19,Z 573.246,A -85,B 0,C 180,E1 -4062.51,E2 -4062.51} C_VEL
LIN {X 0,Y 691.412,Z 451.67,A -85,B 0,C 180,E1 -4063.773,E2 -4063.773} C_VEL
LIN {X 0,Y 690.429,Z 443.737,A -85,B 0,C 180,E1 -4063.886,E2 -4063.886} C_VEL
LIN {X 0,Y 690.73,Z 414.489,A -85,B 0,C 180,E1 -4066.495,E2 -4066.495} C_VEL
LIN {X 0,Y 691.081,Z 384.125,A -85,B 0,C 180,E1 -4069.227,E2 -4069.227} C_VEL
LIN {X 0,Y 691.36,Z 356.892,A -85,B 0,C 180,E1 -4071.703,E2 -4071.703} C_VEL
LIN {X 0,Y 691.626,Z 331.849,A -85,B 0,C 180,E1 -4074.006,E2 -4074.006} C_VEL
LIN {X 0,Y 691.686,Z 321.043,A -85,B 0,C 180,E1 -4075.011,E2 -4075.011} C_VEL
LIN {X 0,Y 690.046,Z 312.092,A -85,B 0,C 180,E1 -4075.92,E2 -4075.92} C_VEL
LIN {X 0,Y 689.986,Z 312.091,A -85,B 0,C 180,E1 -4078.498,E2 -4078.498} C_VEL
LIN {X 0,Y 689.993,Z 312.089,A -85,B 0,C 180,E1 -4080.502,E2 -4080.502} C_VEL
LIN {X 0,Y 689.998,Z 312.088,A -85,B 0,C 180,E1 -4082.588,E2 -4082.588} C_VEL
LIN {X 0,Y 690.004,Z 312.097,A -85,B 0,C 180,E1 -4085.354,E2 -4085.354} C_VEL
LIN {X 0,Y 689.989,Z 312.095,A -85,B 0,C 180,E1 -4087.644,E2 -4087.644} C_VEL
LIN {X 0,Y 690.009,Z 312.087,A -85,B 0,C 180,E1 -4090.517,E2 -4090.517} C_VEL
LIN {X 0,Y 689.974,Z 312.1,A -85,B 0,C 180,E1 -4093.036,E2 -4093.036} C_VEL
LIN {X 0,Y 690.03,Z 312.089,A -85,B 0,C 180,E1 -4095.54,E2 -4095.54} C_VEL
LIN {X 0,Y 689.969,Z 312.092,A -85,B 0,C 180,E1 -4097.931,E2 -4097.931} C_VEL
LIN {X 0,Y 689.99,Z 312.09,A -85,B 0,C 180,E1 -4100.242,E2 -4100.242} C_VEL
LIN {X 0,Y 689.997,Z 312.092,A -85,B 0,C 180,E1 -4102.477,E2 -4102.477} C_VEL
LIN {X 0,Y 690.037,Z 312.092,A -85,B 0,C 180,E1 -4104.648,E2 -4104.648} C_VEL
LIN {X 0,Y 690.044,Z 312.086,A -85,B 0,C 180,E1 -4107.453,E2 -4107.453} C_VEL
LIN {X 0,Y 690.013,Z 312.094,A -85,B 0,C 180,E1 -4110.171,E2 -4110.171} C_VEL
LIN {X 0,Y 689.999,Z 312.098,A -85,B 0,C 180,E1 -4112.818,E2 -4112.818} C_VEL
LIN {X 0,Y 690.075,Z 312.205,A -85,B 0,C 180,E1 -4114.551,E2 -4114.551} C_VEL
LIN {X 0,Y 691.481,Z 320.205,A -85,B 0,C 180,E1 -4115.301,E2 -4115.301} C_VEL
LIN {X 0,Y 691.46,Z 344.924,A -85,B 0,C 180,E1 -4117.517,E2 -4117.517} C_VEL
LIN {X 0,Y 691.251,Z 370.681,A -85,B 0,C 180,E1 -4119.847,E2 -4119.847} C_VEL
LIN {X 0,Y 691.019,Z 396.051,A -85,B 0,C 180,E1 -4122.144,E2 -4122.144} C_VEL
LIN {X 0,Y 690.665,Z 425.247,A -85,B 0,C 180,E1 -4124.862,E2 -4124.862} C_VEL
LIN {X 0,Y 690.501,Z 439.759,A -85,B 0,C 180,E1 -4126.181,E2 -4126.181} C_VEL
LIN {X 0,Y 691.46,Z 447.433,A -85,B 0,C 180,E1 -4126.284,E2 -4126.284} C_VEL
LIN {X 0,Y 691.122,Z 576.716,A -85,B 0,C 180,E1 -4127.637,E2 -4127.637} C_VEL
LIN {X 0,Y 691.037,Z 589.45,A -85,B 0,C 180,E1 -4127.859,E2 -4127.859} C_VEL
LIN {X 0,Y 690.934,Z 600.101,A -85,B 0,C 180,E1 -4128.117,E2 -4128.117} C_VEL
LIN {X 0,Y 690.768,Z 611.756,A -85,B 0,C 180,E1 -4128.485,E2 -4128.485} C_VEL
LIN {X 0,Y 690.564,Z 622.054,A -85,B 0,C 180,E1 -4128.889,E2 -4128.889} C_VEL
LIN {X 0,Y 690.441,Z 631.415,A -85,B 0,C 180,E1 -4129.331,E2 -4129.331} C_VEL
LIN {X 0,Y 690.347,Z 640.635,A -85,B 0,C 180,E1 -4129.844,E2 -4129.844} C_VEL
LIN {X 0,Y 690.216,Z 649.688,A -85,B 0,C 180,E1 -4130.435,E2 -4130.435} C_VEL
LIN {X 0,Y 690.038,Z 658.364,A -85,B 0,C 180,E1 -4131.095,E2 -4131.095} C_VEL
LIN {X 0,Y 689.909,Z 666.594,A -85,B 0,C 180,E1 -4131.829,E2 -4131.829} C_VEL
LIN {X 0,Y 689.814,Z 673.641,A -85,B 0,C 180,E1 -4132.561,E2 -4132.561} C_VEL
LIN {X 0,Y 689.726,Z 679.696,A -85,B 0,C 180,E1 -4133.293,E2 -4133.293} C_VEL
LIN {X 0,Y 689.661,Z 685.829,A -85,B 0,C 180,E1 -4134.171,E2 -4134.171} C_VEL
LIN {X 0,Y 689.643,Z 690.901,A -85,B 0,C 180,E1 -4135.048,E2 -4135.048} C_VEL
LIN {X 0,Y 689.548,Z 695.015,A -85,B 0,C 180,E1 -4135.923,E2 -4135.923} C_VEL
LIN {X 0,Y 689.57,Z 697.332,A -85,B 0,C 180,E1 -4136.506,E2 -4136.506} C_VEL
LIN {X 0,Y 689.542,Z 700.721,A -85,B 0,C 180,E1 -4137.671,E2 -4137.671} C_VEL
LIN {X 0,Y 689.491,Z 702.765,A -85,B 0,C 180,E1 -4138.836,E2 -4138.836} C_VEL
LIN {X 0,Y 689.461,Z 703.494,A -85,B 0,C 180,E1 -4140,E2 -4140} C_VEL
LIN {X 0,Y 689.49,Z 702.854,A -85,B 0,C 180,E1 -4141.164,E2 -4141.164} C_VEL
LIN {X 0,Y 689.541,Z 700.93,A -85,B 0,C 180,E1 -4142.329,E2 -4142.329} C_VEL
LIN {X 0,Y 689.582,Z 699.475,A -85,B 0,C 180,E1 -4142.911,E2 -4142.911} C_VEL
LIN {X 0,Y 689.548,Z 695.389,A -85,B 0,C 180,E1 -4144.078,E2 -4144.078} C_VEL
LIN {X 0,Y 689.641,Z 691.37,A -85,B 0,C 180,E1 -4144.953,E2 -4144.953} C_VEL
LIN {X 0,Y 689.634,Z 686.125,A -85,B 0,C 180,E1 -4145.872,E2 -4145.872} C_VEL
LIN {X 0,Y 689.744,Z 679.27,A -85,B 0,C 180,E1 -4146.853,E2 -4146.853} C_VEL
LIN {X 0,Y 689.852,Z 670.512,A -85,B 0,C 180,E1 -4147.879,E2 -4147.879} C_VEL
LIN {X 0,Y 689.988,Z 661.187,A -85,B 0,C 180,E1 -4148.759,E2 -4148.759} C_VEL
LIN {X 0,Y 690.171,Z 651.951,A -85,B 0,C 180,E1 -4149.493,E2 -4149.493} C_VEL
LIN {X 0,Y 690.271,Z 643.254,A -85,B 0,C 180,E1 -4150.084,E2 -4150.084} C_VEL
LIN {X 0,Y 690.406,Z 634.511,A -85,B 0,C 180,E1 -4150.596,E2 -4150.596} C_VEL
LIN {X 0,Y 690.573,Z 624.084,A -85,B 0,C 180,E1 -4151.112,E2 -4151.112} C_VEL
LIN {X 0,Y 690.767,Z 613.219,A -85,B 0,C 180,E1 -4151.553,E2 -4151.553} C_VEL
LIN {X 0,Y 690.88,Z 603.211,A -85,B 0,C 180,E1 -4151.885,E2 -4151.885} C_VEL
LIN {X 0,Y 690.972,Z 591.863,A -85,B 0,C 180,E1 -4152.18,E2 -4152.18} C_VEL
LIN {X 0,Y 691.102,Z 581.362,A -85,B 0,C 180,E1 -4152.382,E2 -4152.382} C_VEL
LIN {X 0,Y 691.159,Z 567.068,A -85,B 0,C 180,E1 -4152.567,E2 -4152.567} C_VEL
LIN {X 0,Y 691.376,Z 446.283,A -85,B 0,C 180,E1 -4153.82,E2 -4153.82} C_VEL
LIN {X 0,Y 690.475,Z 439.544,A -85,B 0,C 180,E1 -4153.923,E2 -4153.923} C_VEL
LIN {X 0,Y 690.802,Z 415.055,A -85,B 0,C 180,E1 -4156.191,E2 -4156.191} C_VEL
LIN {X 0,Y 690.973,Z 404.22,A -85,B 0,C 180,E1 -4157.204,E2 -4157.204} C_VEL
LIN {X 0,Y 690.413,Z 400.43,A -85,B 0,C 180,E1 -4157.574,E2 -4157.574} C_VEL
LIN {X 0,Y 684.889,Z 388.534,A -85,B 0,C 180,E1 -4158.818,E2 -4158.818} C_VEL
LIN {X 0,Y 684.283,Z 384.685,A -85,B 0,C 180,E1 -4159.193,E2 -4159.193} C_VEL
LIN {X 0,Y 684.663,Z 357.133,A -85,B 0,C 180,E1 -4161.769,E2 -4161.769} C_VEL
LIN {X 0,Y 685.015,Z 330.723,A -85,B 0,C 180,E1 -4164.268,E2 -4164.268} C_VEL
LIN {X 0,Y 685.155,Z 323.595,A -85,B 0,C 180,E1 -4164.943,E2 -4164.943} C_VEL
LIN {X 0,Y 683.008,Z 312.967,A -85,B 0,C 180,E1 -4166.037,E2 -4166.037} C_VEL
LIN {X 0,Y 683.002,Z 312.963,A -85,B 0,C 180,E1 -4168.817,E2 -4168.817} C_VEL
LIN {X 0,Y 683.011,Z 312.965,A -85,B 0,C 180,E1 -4171.535,E2 -4171.535} C_VEL
LIN {X 0,Y 682.987,Z 312.963,A -85,B 0,C 180,E1 -4173.829,E2 -4173.829} C_VEL
LIN {X 0,Y 682.99,Z 312.961,A -85,B 0,C 180,E1 -4176.5,E2 -4176.5} C_VEL
LIN {X 0,Y 682.987,Z 312.966,A -85,B 0,C 180,E1 -4178.792,E2 -4178.792} C_VEL
LIN {X 0,Y 683.009,Z 312.961,A -85,B 0,C 180,E1 -4181.528,E2 -4181.528} C_VEL
LIN {X 0,Y 683.033,Z 312.956,A -85,B 0,C 180,E1 -4184.214,E2 -4184.214} C_VEL
LIN {X 0,Y 683.008,Z 312.967,A -85,B 0,C 180,E1 -4186.73,E2 -4186.73} C_VEL
LIN {X 0,Y 683.03,Z 312.957,A -85,B 0,C 180,E1 -4189.365,E2 -4189.365} C_VEL
LIN {X 0,Y 682.979,Z 312.965,A -85,B 0,C 180,E1 -4192.157,E2 -4192.157} C_VEL
LIN {X 0,Y 683.007,Z 312.964,A -85,B 0,C 180,E1 -4194.229,E2 -4194.229} C_VEL
LIN {X 0,Y 682.995,Z 312.969,A -85,B 0,C 180,E1 -4196.372,E2 -4196.372} C_VEL
LIN {X 0,Y 682.972,Z 312.963,A -85,B 0,C 180,E1 -4199.15,E2 -4199.15} C_VEL
LIN {X 0,Y 683.028,Z 312.96,A -85,B 0,C 180,E1 -4201.877,E2 -4201.877} C_VEL
LIN {X 0,Y 683,Z 312.965,A -85,B 0,C 180,E1 -4204.486,E2 -4204.486} C_VEL
LIN {X 0,Y 683.018,Z 312.958,A -85,B 0,C 180,E1 -4207.364,E2 -4207.364} C_VEL
LIN {X 0,Y 682.982,Z 312.966,A -85,B 0,C 180,E1 -4209.593,E2 -4209.593} C_VEL
LIN {X 0,Y 683.014,Z 312.961,A -85,B 0,C 180,E1 -4211.463,E2 -4211.463} C_VEL
LIN {X 0,Y 683,Z 312.97,A -85,B 0,C 180,E1 -4213.925,E2 -4213.925} C_VEL
LIN {X 0,Y 682.993,Z 312.962,A -85,B 0,C 180,E1 -4216.357,E2 -4216.357} C_VEL
LIN {X 0,Y 683.008,Z 312.959,A -85,B 0,C 180,E1 -4218.764,E2 -4218.764} C_VEL
LIN {X 0,Y 683.041,Z 312.955,A -85,B 0,C 180,E1 -4220.556,E2 -4220.556} C_VEL
LIN {X 0,Y 683.018,Z 313.141,A -85,B 0,C 180,E1 -4221.17,E2 -4221.17} C_VEL
LIN {X 0,Y 684.663,Z 319.079,A -85,B 0,C 180,E1 -4221.269,E2 -4221.269} C_VEL
LIN {X 0,Y 684.34,Z 436.42,A -85,B 0,C 180,E1 -4222.52,E2 -4222.52} C_VEL
LIN {X 0,Y 684.286,Z 449.535,A -85,B 0,C 180,E1 -4222.76,E2 -4222.76} C_VEL
LIN {X 0,Y 684.137,Z 463.379,A -85,B 0,C 180,E1 -4223.128,E2 -4223.128} C_VEL
LIN {X 0,Y 683.979,Z 477.482,A -85,B 0,C 180,E1 -4223.643,E2 -4223.643} C_VEL
LIN {X 0,Y 683.766,Z 490.669,A -85,B 0,C 180,E1 -4224.268,E2 -4224.268} C_VEL
LIN {X 0,Y 683.603,Z 501.908,A -85,B 0,C 180,E1 -4224.93,E2 -4224.93} C_VEL
LIN {X 0,Y 683.376,Z 511.292,A -85,B 0,C 180,E1 -4225.591,E2 -4225.591} C_VEL
LIN {X 0,Y 683.231,Z 520.112,A -85,B 0,C 180,E1 -4226.326,E2 -4226.326} C_VEL
LIN {X 0,Y 683.064,Z 527.666,A -85,B 0,C 180,E1 -4227.061,E2 -4227.061} C_VEL
LIN {X 0,Y 682.903,Z 535.294,A -85,B 0,C 180,E1 -4227.943,E2 -4227.943} C_VEL
LIN {X 0,Y 682.737,Z 541.673,A -85,B 0,C 180,E1 -4228.824,E2 -4228.824} C_VEL
LIN {X 0,Y 682.727,Z 546.939,A -85,B 0,C 180,E1 -4229.706,E2 -4229.706} C_VEL
LIN {X 0,Y 682.613,Z 551.285,A -85,B 0,C 180,E1 -4230.588,E2 -4230.588} C_VEL
LIN {X 0,Y 682.539,Z 555.659,A -85,B 0,C 180,E1 -4231.764,E2 -4231.764} C_VEL
LIN {X 0,Y 682.575,Z 557.37,A -85,B 0,C 180,E1 -4232.353,E2 -4232.353} C_VEL
LIN {X 0,Y 682.573,Z 559.682,A -85,B 0,C 180,E1 -4233.53,E2 -4233.53} C_VEL
LIN {X 0,Y 682.548,Z 560.69,A -85,B 0,C 180,E1 -4234.709,E2 -4234.709} C_VEL
LIN {X 0,Y 682.572,Z 560.395,A -85,B 0,C 180,E1 -4235.89,E2 -4235.89} C_VEL
LIN {X 0,Y 682.578,Z 559.794,A -85,B 0,C 180,E1 -4236.481,E2 -4236.481} C_VEL
LIN {X 0,Y 682.587,Z 557.557,A -85,B 0,C 180,E1 -4237.666,E2 -4237.666} C_VEL
LIN {X 0,Y 682.636,Z 553.913,A -85,B 0,C 180,E1 -4238.854,E2 -4238.854} C_VEL
LIN {X 0,Y 682.711,Z 548.713,A -85,B 0,C 180,E1 -4240.045,E2 -4240.045} C_VEL
LIN {X 0,Y 682.796,Z 543.743,A -85,B 0,C 180,E1 -4240.94,E2 -4240.94} C_VEL
LIN {X 0,Y 682.905,Z 537.682,A -85,B 0,C 180,E1 -4241.838,E2 -4241.838} C_VEL
LIN {X 0,Y 683.057,Z 530.571,A -85,B 0,C 180,E1 -4242.712,E2 -4242.712} C_VEL
LIN {X 0,Y 683.175,Z 523.278,A -85,B 0,C 180,E1 -4243.474,E2 -4243.474} C_VEL
LIN {X 0,Y 683.339,Z 514.614,A -85,B 0,C 180,E1 -4244.242,E2 -4244.242} C_VEL
LIN {X 0,Y 683.501,Z 504.445,A -85,B 0,C 180,E1 -4244.997,E2 -4244.997} C_VEL
LIN {X 0,Y 683.667,Z 494.428,A -85,B 0,C 180,E1 -4245.619,E2 -4245.619} C_VEL
LIN {X 0,Y 683.888,Z 482.971,A -85,B 0,C 180,E1 -4246.206,E2 -4246.206} C_VEL
LIN {X 0,Y 684.058,Z 471.065,A -85,B 0,C 180,E1 -4246.699,E2 -4246.699} C_VEL
LIN {X 0,Y 684.205,Z 458.122,A -85,B 0,C 180,E1 -4247.117,E2 -4247.117} C_VEL
LIN {X 0,Y 684.282,Z 444.639,A -85,B 0,C 180,E1 -4247.435,E2 -4247.435} C_VEL
LIN {X 0,Y 684.368,Z 430.328,A -85,B 0,C 180,E1 -4247.65,E2 -4247.65} C_VEL
LIN {X 0,Y 684.533,Z 318.034,A -85,B 0,C 180,E1 -4248.835,E2 -4248.835} C_VEL
LIN {X 0,Y 682.985,Z 312.969,A -85,B 0,C 180,E1 -4248.939,E2 -4248.939} C_VEL
LIN {X 0,Y 682.97,Z 312.967,A -85,B 0,C 180,E1 -4251.667,E2 -4251.667} C_VEL
LIN {X 0,Y 682.959,Z 312.975,A -85,B 0,C 180,E1 -4254.22,E2 -4254.22} C_VEL
LIN {X 0,Y 682.973,Z 312.968,A -85,B 0,C 180,E1 -4256.841,E2 -4256.841} C_VEL
LIN {X 0,Y 682.966,Z 312.964,A -85,B 0,C 180,E1 -4259.491,E2 -4259.491} C_VEL
LIN {X 0,Y 682.949,Z 312.976,A -85,B 0,C 180,E1 -4262.23,E2 -4262.23} C_VEL
LIN {X 0,Y 682.963,Z 312.964,A -85,B 0,C 180,E1 -4265.053,E2 -4265.053} C_VEL
LIN {X 0,Y 682.97,Z 312.97,A -85,B 0,C 180,E1 -4267.978,E2 -4267.978} C_VEL
LIN {X 0,Y 682.975,Z 312.966,A -85,B 0,C 180,E1 -4270.63,E2 -4270.63} C_VEL
LIN {X 0,Y 682.94,Z 312.968,A -85,B 0,C 180,E1 -4273.407,E2 -4273.407} C_VEL
LIN {X 0,Y 682.988,Z 312.968,A -85,B 0,C 180,E1 -4275.881,E2 -4275.881} C_VEL
LIN {X 0,Y 682.964,Z 312.967,A -85,B 0,C 180,E1 -4278.477,E2 -4278.477} C_VEL
LIN {X 0,Y 682.976,Z 312.962,A -85,B 0,C 180,E1 -4281.273,E2 -4281.273} C_VEL
LIN {X 0,Y 682.968,Z 312.967,A -85,B 0,C 180,E1 -4284.117,E2 -4284.117} C_VEL
LIN {X 0,Y 682.979,Z 312.964,A -85,B 0,C 180,E1 -4286.371,E2 -4286.371} C_VEL
LIN {X 0,Y 682.993,Z 312.959,A -85,B 0,C 180,E1 -4288.464,E2 -4288.464} C_VEL
LIN {X 0,Y 682.95,Z 312.966,A -85,B 0,C 180,E1 -4291.181,E2 -4291.181} C_VEL
LIN {X 0,Y 682.932,Z 312.975,A -85,B 0,C 180,E1 -4293.83,E2 -4293.83} C_VEL
LIN {X 0,Y 682.982,Z 312.969,A -85,B 0,C 180,E1 -4295.89,E2 -4295.89} C_VEL
LIN {X 0,Y 682.965,Z 312.963,A -85,B 0,C 180,E1 -4298.333,E2 -4298.333} C_VEL
LIN {X 0,Y 682.979,Z 312.964,A -85,B 0,C 180,E1 -4300.841,E2 -4300.841} C_VEL
LIN {X 0,Y 682.976,Z 312.971,A -85,B 0,C 180,E1 -4303.312,E2 -4303.312} C_VEL
LIN {X 0,Y 682.986,Z 312.969,A -85,B 0,C 180,E1 -4305.201,E2 -4305.201} C_VEL
LIN {X 0,Y 684.439,Z 317.744,A -85,B 0,C 180,E1 -4305.29,E2 -4305.29} C_VEL
LIN {X 0,Y 684.205,Z 434.923,A -85,B 0,C 180,E1 -4306.561,E2 -4306.561} C_VEL
LIN {X 0,Y 684.065,Z 448.855,A -85,B 0,C 180,E1 -4306.82,E2 -4306.82} C_VEL
LIN {X 0,Y 683.914,Z 462.863,A -85,B 0,C 180,E1 -4307.204,E2 -4307.204} C_VEL
LIN {X 0,Y 683.74,Z 475.157,A -85,B 0,C 180,E1 -4307.652,E2 -4307.652} C_VEL
LIN {X 0,Y 683.597,Z 486.593,A -85,B 0,C 180,E1 -4308.174,E2 -4308.174} C_VEL
LIN {X 0,Y 683.381,Z 497.325,A -85,B 0,C 180,E1 -4308.77,E2 -4308.77} C_VEL
LIN {X 0,Y 683.249,Z 507.479,A -85,B 0,C 180,E1 -4309.448,E2 -4309.448} C_VEL
LIN {X 0,Y 683.072,Z 515.935,A -85,B 0,C 180,E1 -4310.114,E2 -4310.114} C_VEL
LIN {X 0,Y 682.986,Z 523.934,A -85,B 0,C 180,E1 -4310.853,E2 -4310.853} C_VEL
LIN {X 0,Y 682.841,Z 530.824,A -85,B 0,C 180,E1 -4311.595,E2 -4311.595} C_VEL
LIN {X 0,Y 682.703,Z 537.787,A -85,B 0,C 180,E1 -4312.483,E2 -4312.483} C_VEL
LIN {X 0,Y 682.642,Z 542.707,A -85,B 0,C 180,E1 -4313.223,E2 -4313.223} C_VEL
LIN {X 0,Y 682.571,Z 547.632,A -85,B 0,C 180,E1 -4314.11,E2 -4314.11} C_VEL
LIN {X 0,Y 682.575,Z 552.659,A -85,B 0,C 180,E1 -4315.291,E2 -4315.291} C_VEL
LIN {X 0,Y 682.477,Z 554.706,A -85,B 0,C 180,E1 -4315.88,E2 -4315.88} C_VEL
LIN {X 0,Y 682.514,Z 557.584,A -85,B 0,C 180,E1 -4317.058,E2 -4317.058} C_VEL
LIN {X 0,Y 682.466,Z 559.115,A -85,B 0,C 180,E1 -4318.235,E2 -4318.235} C_VEL
LIN {X 0,Y 682.414,Z 559.347,A -85,B 0,C 180,E1 -4319.412,E2 -4319.412} C_VEL
LIN {X 0,Y 682.406,Z 559.045,A -85,B 0,C 180,E1 -4320,E2 -4320} C_VEL
LIN {X 0,Y 682.441,Z 557.364,A -85,B 0,C 180,E1 -4321.176,E2 -4321.176} C_VEL
LIN {X 0,Y 682.544,Z 554.286,A -85,B 0,C 180,E1 -4322.352,E2 -4322.352} C_VEL
LIN {X 0,Y 682.564,Z 551.118,A -85,B 0,C 180,E1 -4323.235,E2 -4323.235} C_VEL
LIN {X 0,Y 682.599,Z 545.433,A -85,B 0,C 180,E1 -4324.414,E2 -4324.414} C_VEL
LIN {X 0,Y 682.743,Z 540.076,A -85,B 0,C 180,E1 -4325.298,E2 -4325.298} C_VEL
LIN {X 0,Y 682.845,Z 533.601,A -85,B 0,C 180,E1 -4326.183,E2 -4326.183} C_VEL
LIN {X 0,Y 682.95,Z 525.801,A -85,B 0,C 180,E1 -4327.069,E2 -4327.069} C_VEL
LIN {X 0,Y 683.078,Z 518.104,A -85,B 0,C 180,E1 -4327.809,E2 -4327.809} C_VEL
LIN {X 0,Y 683.293,Z 507.988,A -85,B 0,C 180,E1 -4328.622,E2 -4328.622} C_VEL
LIN {X 0,Y 683.439,Z 498.069,A -85,B 0,C 180,E1 -4329.289,E2 -4329.289} C_VEL
LIN {X 0,Y 683.645,Z 487.489,A -85,B 0,C 180,E1 -4329.882,E2 -4329.882} C_VEL
LIN {X 0,Y 683.786,Z 476.034,A -85,B 0,C 180,E1 -4330.411,E2 -4330.411} C_VEL
LIN {X 0,Y 683.938,Z 463.092,A -85,B 0,C 180,E1 -4330.884,E2 -4330.884} C_VEL
LIN {X 0,Y 684.049,Z 448.743,A -85,B 0,C 180,E1 -4331.275,E2 -4331.275} C_VEL
LIN {X 0,Y 684.215,Z 434.056,A -85,B 0,C 180,E1 -4331.534,E2 -4331.534} C_VEL
LIN {X 0,Y 684.493,Z 317.756,A -85,B 0,C 180,E1 -4332.797,E2 -4332.797} C_VEL
LIN {X 0,Y 683.078,Z 312.957,A -85,B 0,C 180,E1 -4332.886,E2 -4332.886} C_VEL
LIN {X 0,Y 683.05,Z 312.955,A -85,B 0,C 180,E1 -4335.463,E2 -4335.463} C_VEL
LIN {X 0,Y 683.013,Z 312.966,A -85,B 0,C 180,E1 -4337.918,E2 -4337.918} C_VEL
LIN {X 0,Y 682.982,Z 312.968,A -85,B 0,C 180,E1 -4339.782,E2 -4339.782} C_VEL
LIN {X 0,Y 683.012,Z 312.967,A -85,B 0,C 180,E1 -4342.299,E2 -4342.299} C_VEL
LIN {X 0,Y 683.002,Z 312.96,A -85,B 0,C 180,E1 -4344.864,E2 -4344.864} C_VEL
LIN {X 0,Y 682.984,Z 312.967,A -85,B 0,C 180,E1 -4347.484,E2 -4347.484} C_VEL
LIN {X 0,Y 682.989,Z 312.967,A -85,B 0,C 180,E1 -4349.49,E2 -4349.49} C_VEL
LIN {X 0,Y 682.987,Z 312.971,A -85,B 0,C 180,E1 -4351.655,E2 -4351.655} C_VEL
LIN {X 0,Y 682.998,Z 312.96,A -85,B 0,C 180,E1 -4354.336,E2 -4354.336} C_VEL
LIN {X 0,Y 682.957,Z 312.966,A -85,B 0,C 180,E1 -4356.872,E2 -4356.872} C_VEL
LIN {X 0,Y 682.96,Z 312.971,A -85,B 0,C 180,E1 -4359.485,E2 -4359.485} C_VEL
LIN {X 0,Y 682.964,Z 312.965,A -85,B 0,C 180,E1 -4361.808,E2 -4361.808} C_VEL
LIN {X 0,Y 682.99,Z 312.959,A -85,B 0,C 180,E1 -4364.217,E2 -4364.217} C_VEL
LIN {X 0,Y 682.94,Z 312.972,A -85,B 0,C 180,E1 -4366.736,E2 -4366.736} C_VEL
LIN {X 0,Y 682.974,Z 312.966,A -85,B 0,C 180,E1 -4369.37,E2 -4369.37} C_VEL
LIN {X 0,Y 682.972,Z 312.964,A -85,B 0,C 180,E1 -4372.022,E2 -4372.022} C_VEL
LIN {X 0,Y 682.959,Z 312.969,A -85,B 0,C 180,E1 -4374.946,E2 -4374.946} C_VEL
LIN {X 0,Y 682.973,Z 312.965,A -85,B 0,C 180,E1 -4377.243,E2 -4377.243} C_VEL
LIN {X 0,Y 682.951,Z 312.968,A -85,B 0,C 180,E1 -4379.831,E2 -4379.831} C_VEL
LIN {X 0,Y 682.952,Z 312.976,A -85,B 0,C 180,E1 -4382.514,E2 -4382.514} C_VEL
LIN {X 0,Y 682.981,Z 313.004,A -85,B 0,C 180,E1 -4383.982,E2 -4383.982} C_VEL
LIN {X 0,Y 684.713,Z 321.881,A -85,B 0,C 180,E1 -4384.879,E2 -4384.879} C_VEL
LIN {X 0,Y 684.591,Z 340.852,A -85,B 0,C 180,E1 -4386.658,E2 -4386.658} C_VEL
LIN {X 0,Y 684.275,Z 369.653,A -85,B 0,C 180,E1 -4389.32,E2 -4389.32} C_VEL
LIN {X 0,Y 683.905,Z 398.464,A -85,B 0,C 180,E1 -4391.952,E2 -4391.952} C_VEL
LIN {X 0,Y 683.529,Z 427.163,A -85,B 0,C 180,E1 -4394.548,E2 -4394.548} C_VEL
LIN {X 0,Y 683.384,Z 442.931,A -85,B 0,C 180,E1 -4395.968,E2 -4395.968} C_VEL
LIN {X 0,Y 684.595,Z 454.444,A -85,B 0,C 180,E1 -4396.125,E2 -4396.125} C_VEL
LIN {X 0,Y 684.152,Z 581.913,A -85,B 0,C 180,E1 -4397.472,E2 -4397.472} C_VEL
LIN {X 0,Y 684,Z 596.006,A -85,B 0,C 180,E1 -4397.732,E2 -4397.732} C_VEL
LIN {X 0,Y 683.892,Z 609.75,A -85,B 0,C 180,E1 -4398.105,E2 -4398.105} C_VEL
LIN {X 0,Y 683.695,Z 622.231,A -85,B 0,C 180,E1 -4398.551,E2 -4398.551} C_VEL
LIN {X 0,Y 683.467,Z 635.301,A -85,B 0,C 180,E1 -4399.145,E2 -4399.145} C_VEL
LIN {X 0,Y 683.268,Z 647.704,A -85,B 0,C 180,E1 -4399.848,E2 -4399.848} C_VEL
LIN {X 0,Y 683.085,Z 658.062,A -85,B 0,C 180,E1 -4400.557,E2 -4400.557} C_VEL
LIN {X 0,Y 682.904,Z 668.854,A -85,B 0,C 180,E1 -4401.447,E2 -4401.447} C_VEL
LIN {X 0,Y 682.768,Z 677.756,A -85,B 0,C 180,E1 -4402.336,E2 -4402.336} C_VEL
LIN {X 0,Y 682.655,Z 685.09,A -85,B 0,C 180,E1 -4403.223,E2 -4403.223} C_VEL
LIN {X 0,Y 682.558,Z 692.388,A -85,B 0,C 180,E1 -4404.309,E2 -4404.309} C_VEL
LIN {X 0,Y 682.53,Z 697.643,A -85,B 0,C 180,E1 -4405.291,E2 -4405.291} C_VEL
LIN {X 0,Y 682.47,Z 702.489,A -85,B 0,C 180,E1 -4406.469,E2 -4406.469} C_VEL
LIN {X 0,Y 682.455,Z 705.855,A -85,B 0,C 180,E1 -4407.647,E2 -4407.647} C_VEL
LIN {X 0,Y 682.41,Z 707.842,A -85,B 0,C 180,E1 -4408.824,E2 -4408.824} C_VEL
LIN {X 0,Y 682.378,Z 708.5,A -85,B 0,C 180,E1 -4410,E2 -4410} C_VEL
LIN {X 0,Y 682.41,Z 707.84,A -85,B 0,C 180,E1 -4411.176,E2 -4411.176} C_VEL
LIN {X 0,Y 682.455,Z 705.852,A -85,B 0,C 180,E1 -4412.353,E2 -4412.353} C_VEL
LIN {X 0,Y 682.47,Z 702.486,A -85,B 0,C 180,E1 -4413.53,E2 -4413.53} C_VEL
LIN {X 0,Y 682.53,Z 697.646,A -85,B 0,C 180,E1 -4414.709,E2 -4414.709} C_VEL
LIN {X 0,Y 682.569,Z 692.98,A -85,B 0,C 180,E1 -4415.594,E2 -4415.594} C_VEL
LIN {X 0,Y 682.64,Z 686.202,A -85,B 0,C 180,E1 -4416.629,E2 -4416.629} C_VEL
LIN {X 0,Y 682.749,Z 679.116,A -85,B 0,C 180,E1 -4417.516,E2 -4417.516} C_VEL
LIN {X 0,Y 682.874,Z 670.5,A -85,B 0,C 180,E1 -4418.405,E2 -4418.405} C_VEL
LIN {X 0,Y 683.073,Z 660.043,A -85,B 0,C 180,E1 -4419.294,E2 -4419.294} C_VEL
LIN {X 0,Y 683.25,Z 649.557,A -85,B 0,C 180,E1 -4420.037,E2 -4420.037} C_VEL
LIN {X 0,Y 683.432,Z 638.186,A -85,B 0,C 180,E1 -4420.706,E2 -4420.706} C_VEL
LIN {X 0,Y 683.635,Z 625.801,A -85,B 0,C 180,E1 -4421.3,E2 -4421.3} C_VEL
LIN {X 0,Y 683.874,Z 612.053,A -85,B 0,C 180,E1 -4421.82,E2 -4421.82} C_VEL
LIN {X 0,Y 684.019,Z 598.34,A -85,B 0,C 180,E1 -4422.212,E2 -4422.212} C_VEL
LIN {X 0,Y 684.174,Z 584.285,A -85,B 0,C 180,E1 -4422.49,E2 -4422.49} C_VEL
LIN {X 0,Y 684.288,Z 559.956,A -85,B 0,C 180,E1 -4422.77,E2 -4422.77} C_VEL
LIN {X 0,Y 684.455,Z 452.016,A -85,B 0,C 180,E1 -4423.904,E2 -4423.904} C_VEL
LIN {X 0,Y 683.385,Z 442.959,A -85,B 0,C 180,E1 -4424.032,E2 -4424.032} C_VEL
LIN {X 0,Y 683.735,Z 413.713,A -85,B 0,C 180,E1 -4426.669,E2 -4426.669} C_VEL
LIN {X 0,Y 684.073,Z 383.946,A -85,B 0,C 180,E1 -4429.377,E2 -4429.377} C_VEL
LIN {X 0,Y 684.399,Z 357.818,A -85,B 0,C 180,E1 -4431.777,E2 -4431.777} C_VEL
LIN {X 0,Y 684.67,Z 333.953,A -85,B 0,C 180,E1 -4433.995,E2 -4433.995} C_VEL
LIN {X 0,Y 684.708,Z 321.959,A -85,B 0,C 180,E1 -4435.121,E2 -4435.121} C_VEL
LIN {X 0,Y 682.999,Z 312.97,A -85,B 0,C 180,E1 -4436.037,E2 -4436.037} C_VEL
LIN {X 0,Y 682.948,Z 312.968,A -85,B 0,C 180,E1 -4438.819,E2 -4438.819} C_VEL
LIN {X 0,Y 682.979,Z 312.973,A -85,B 0,C 180,E1 -4441.537,E2 -4441.537} C_VEL
LIN {X 0,Y 682.948,Z 312.971,A -85,B 0,C 180,E1 -4443.824,E2 -4443.824} C_VEL
LIN {X 0,Y 682.936,Z 312.968,A -85,B 0,C 180,E1 -4446.503,E2 -4446.503} C_VEL
LIN {X 0,Y 682.936,Z 312.97,A -85,B 0,C 180,E1 -4448.787,E2 -4448.787} C_VEL
LIN {X 0,Y 682.96,Z 312.971,A -85,B 0,C 180,E1 -4451.523,E2 -4451.523} C_VEL
LIN {X 0,Y 682.981,Z 312.963,A -85,B 0,C 180,E1 -4454.218,E2 -4454.218} C_VEL
LIN {X 0,Y 682.932,Z 312.974,A -85,B 0,C 180,E1 -4456.736,E2 -4456.736} C_VEL
LIN {X 0,Y 682.972,Z 312.968,A -85,B 0,C 180,E1 -4459.37,E2 -4459.37} C_VEL
LIN {X 0,Y 682.966,Z 312.964,A -85,B 0,C 180,E1 -4462.158,E2 -4462.158} C_VEL
LIN {X 0,Y 682.981,Z 312.972,A -85,B 0,C 180,E1 -4464.948,E2 -4464.948} C_VEL
LIN {X 0,Y 682.988,Z 312.967,A -85,B 0,C 180,E1 -4467.242,E2 -4467.242} C_VEL
LIN {X 0,Y 682.954,Z 312.971,A -85,B 0,C 180,E1 -4469.831,E2 -4469.831} C_VEL
LIN {X 0,Y 682.961,Z 312.976,A -85,B 0,C 180,E1 -4472.515,E2 -4472.515} C_VEL
LIN {X 0,Y 683.021,Z 313.085,A -85,B 0,C 180,E1 -4474.427,E2 -4474.427} C_VEL
LIN {X 0,Y 684.536,Z 321.141,A -85,B 0,C 180,E1 -4475.195,E2 -4475.195} C_VEL
LIN {X 0,Y 684.537,Z 344.225,A -85,B 0,C 180,E1 -4477.277,E2 -4477.277} C_VEL
LIN {X 0,Y 684.304,Z 368.459,A -85,B 0,C 180,E1 -4479.477,E2 -4479.477} C_VEL
LIN {X 0,Y 684.085,Z 395.781,A -85,B 0,C 180,E1 -4481.957,E2 -4481.957} C_VEL
LIN {X 0,Y 683.648,Z 426.63,A -85,B 0,C 180,E1 -4484.855,E2 -4484.855} C_VEL
LIN {X 0,Y 683.535,Z 439.699,A -85,B 0,C 180,E1 -4486.037,E2 -4486.037} C_VEL
LIN {X 0,Y 684.584,Z 449.004,A -85,B 0,C 180,E1 -4486.163,E2 -4486.163} C_VEL
LIN {X 0,Y 684.164,Z 576.887,A -85,B 0,C 180,E1 -4487.528,E2 -4487.528} C_VEL
LIN {X 0,Y 684.077,Z 589.562,A -85,B 0,C 180,E1 -4487.752,E2 -4487.752} C_VEL
LIN {X 0,Y 683.935,Z 600.838,A -85,B 0,C 180,E1 -4488.031,E2 -4488.031} C_VEL
LIN {X 0,Y 683.762,Z 612.352,A -85,B 0,C 180,E1 -4488.402,E2 -4488.402} C_VEL
LIN {X 0,Y 683.542,Z 623.381,A -85,B 0,C 180,E1 -4488.848,E2 -4488.848} C_VEL
LIN {X 0,Y 683.395,Z 633.965,A -85,B 0,C 180,E1 -4489.369,E2 -4489.369} C_VEL
LIN {X 0,Y 683.225,Z 645.268,A -85,B 0,C 180,E1 -4490.038,E2 -4490.038} C_VEL
LIN {X 0,Y 683.039,Z 656.531,A -85,B 0,C 180,E1 -4490.854,E2 -4490.854} C_VEL
LIN {X 0,Y 682.887,Z 665.045,A -85,B 0,C 180,E1 -4491.595,E2 -4491.595} C_VEL
LIN {X 0,Y 682.777,Z 672.327,A -85,B 0,C 180,E1 -4492.336,E2 -4492.336} C_VEL
LIN {X 0,Y 682.658,Z 679.69,A -85,B 0,C 180,E1 -4493.224,E2 -4493.224} C_VEL
LIN {X 0,Y 682.602,Z 685.825,A -85,B 0,C 180,E1 -4494.11,E2 -4494.11} C_VEL
LIN {X 0,Y 682.561,Z 690.895,A -85,B 0,C 180,E1 -4494.996,E2 -4494.996} C_VEL
LIN {X 0,Y 682.468,Z 695.012,A -85,B 0,C 180,E1 -4495.88,E2 -4495.88} C_VEL
LIN {X 0,Y 682.471,Z 697.327,A -85,B 0,C 180,E1 -4496.47,E2 -4496.47} C_VEL
LIN {X 0,Y 682.456,Z 700.719,A -85,B 0,C 180,E1 -4497.647,E2 -4497.647} C_VEL
LIN {X 0,Y 682.414,Z 702.762,A -85,B 0,C 180,E1 -4498.824,E2 -4498.824} C_VEL
LIN {X 0,Y 682.377,Z 703.494,A -85,B 0,C 180,E1 -4500,E2 -4500} C_VEL
LIN {X 0,Y 682.412,Z 702.85,A -85,B 0,C 180,E1 -4501.176,E2 -4501.176} C_VEL
LIN {X 0,Y 682.455,Z 700.926,A -85,B 0,C 180,E1 -4502.353,E2 -4502.353} C_VEL
LIN {X 0,Y 682.507,Z 699.468,A -85,B 0,C 180,E1 -4502.942,E2 -4502.942} C_VEL
LIN {X 0,Y 682.468,Z 695.382,A -85,B 0,C 180,E1 -4504.12,E2 -4504.12} C_VEL
LIN {X 0,Y 682.559,Z 691.359,A -85,B 0,C 180,E1 -4505.004,E2 -4505.004} C_VEL
LIN {X 0,Y 682.56,Z 686.386,A -85,B 0,C 180,E1 -4505.89,E2 -4505.89} C_VEL
LIN {X 0,Y 682.656,Z 680.356,A -85,B 0,C 180,E1 -4506.777,E2 -4506.777} C_VEL
LIN {X 0,Y 682.728,Z 674.407,A -85,B 0,C 180,E1 -4507.516,E2 -4507.516} C_VEL
LIN {X 0,Y 682.834,Z 667.474,A -85,B 0,C 180,E1 -4508.257,E2 -4508.257} C_VEL
LIN {X 0,Y 683.004,Z 659.362,A -85,B 0,C 180,E1 -4508.998,E2 -4508.998} C_VEL
LIN {X 0,Y 683.145,Z 650.822,A -85,B 0,C 180,E1 -4509.666,E2 -4509.666} C_VEL
LIN {X 0,Y 683.28,Z 641.793,A -85,B 0,C 180,E1 -4510.27,E2 -4510.27} C_VEL
LIN {X 0,Y 683.444,Z 631.483,A -85,B 0,C 180,E1 -4510.855,E2 -4510.855} C_VEL
LIN {X 0,Y 683.653,Z 620.443,A -85,B 0,C 180,E1 -4511.375,E2 -4511.375} C_VEL
LIN {X 0,Y 683.872,Z 606.537,A -85,B 0,C 180,E1 -4511.896,E2 -4511.896} C_VEL
LIN {X 0,Y 684.009,Z 592.936,A -85,B 0,C 180,E1 -4512.268,E2 -4512.268} C_VEL
LIN {X 0,Y 684.133,Z 580.557,A -85,B 0,C 180,E1 -4512.51,E2 -4512.51} C_VEL
LIN {X 0,Y 684.26,Z 562.379,A -85,B 0,C 180,E1 -4512.733,E2 -4512.733} C_VEL
LIN {X 0,Y 684.49,Z 446.959,A -85,B 0,C 180,E1 -4513.953,E2 -4513.953} C_VEL
LIN {X 0,Y 683.497,Z 439.538,A -85,B 0,C 180,E1 -4514.068,E2 -4514.068} C_VEL
LIN {X 0,Y 683.847,Z 414.906,A -85,B 0,C 180,E1 -4516.36,E2 -4516.36} C_VEL
LIN {X 0,Y 684.222,Z 388.764,A -85,B 0,C 180,E1 -4518.813,E2 -4518.813} C_VEL
LIN {X 0,Y 684.283,Z 384.685,A -85,B 0,C 180,E1 -4519.193,E2 -4519.193} C_VEL
LIN {X 0,Y 683.685,Z 380.865,A -85,B 0,C 180,E1 -4519.567,E2 -4519.567} C_VEL
LIN {X 0,Y 678.223,Z 369.068,A -85,B 0,C 180,E1 -4520.83,E2 -4520.83} C_VEL
LIN {X 0,Y 677.651,Z 365.22,A -85,B 0,C 180,E1 -4521.209,E2 -4521.209} C_VEL
LIN {X 0,Y 678.02,Z 338.31,A -85,B 0,C 180,E1 -4523.76,E2 -4523.76} C_VEL
LIN {X 0,Y 678.245,Z 324.813,A -85,B 0,C 180,E1 -4525.051,E2 -4525.051} C_VEL
LIN {X 0,Y 675.95,Z 313.845,A -85,B 0,C 180,E1 -4526.191,E2 -4526.191} C_VEL
LIN {X 0,Y 675.959,Z 313.839,A -85,B 0,C 180,E1 -4528.468,E2 -4528.468} C_VEL
LIN {X 0,Y 675.97,Z 313.844,A -85,B 0,C 180,E1 -4531.205,E2 -4531.205} C_VEL
LIN {X 0,Y 675.966,Z 313.836,A -85,B 0,C 180,E1 -4534.025,E2 -4534.025} C_VEL
LIN {X 0,Y 675.945,Z 313.838,A -85,B 0,C 180,E1 -4536.204,E2 -4536.204} C_VEL
LIN {X 0,Y 675.938,Z 313.848,A -85,B 0,C 180,E1 -4538.996,E2 -4538.996} C_VEL
LIN {X 0,Y 675.977,Z 313.835,A -85,B 0,C 180,E1 -4541.75,E2 -4541.75} C_VEL
LIN {X 0,Y 675.991,Z 313.835,A -85,B 0,C 180,E1 -4544.36,E2 -4544.36} C_VEL
LIN {X 0,Y 675.952,Z 313.848,A -85,B 0,C 180,E1 -4546.85,E2 -4546.85} C_VEL
LIN {X 0,Y 675.973,Z 313.837,A -85,B 0,C 180,E1 -4549.246,E2 -4549.246} C_VEL
LIN {X 0,Y 675.944,Z 313.839,A -85,B 0,C 180,E1 -4551.957,E2 -4551.957} C_VEL
LIN {X 0,Y 675.953,Z 313.848,A -85,B 0,C 180,E1 -4554.529,E2 -4554.529} C_VEL
LIN {X 0,Y 675.952,Z 313.839,A -85,B 0,C 180,E1 -4557.072,E2 -4557.072} C_VEL
LIN {X 0,Y 675.98,Z 313.834,A -85,B 0,C 180,E1 -4559.487,E2 -4559.487} C_VEL
LIN {X 0,Y 675.951,Z 313.847,A -85,B 0,C 180,E1 -4562.205,E2 -4562.205} C_VEL
LIN {X 0,Y 675.944,Z 313.84,A -85,B 0,C 180,E1 -4564.858,E2 -4564.858} C_VEL
LIN {X 0,Y 675.983,Z 313.835,A -85,B 0,C 180,E1 -4567.456,E2 -4567.456} C_VEL
LIN {X 0,Y 675.943,Z 313.849,A -85,B 0,C 180,E1 -4570.004,E2 -4570.004} C_VEL
LIN {X 0,Y 675.963,Z 313.838,A -85,B 0,C 180,E1 -4572.512,E2 -4572.512} C_VEL
LIN {X 0,Y 675.949,Z 313.838,A -85,B 0,C 180,E1 -4574.986,E2 -4574.986} C_VEL
LIN {X 0,Y 675.986,Z 313.839,A -85,B 0,C 180,E1 -4577.432,E2 -4577.432} C_VEL
LIN {X 0,Y 676.035,Z 313.834,A -85,B 0,C 180,E1 -4579.855,E2 -4579.855} C_VEL
LIN {X 0,Y 675.96,Z 313.839,A -85,B 0,C 180,E1 -4581.021,E2 -4581.021} C_VEL
LIN {X 0,Y 677.707,Z 319.442,A -85,B 0,C 180,E1 -4581.12,E2 -4581.12} C_VEL
LIN {X 0,Y 677.456,Z 437.043,A -85,B 0,C 180,E1 -4582.388,E2 -4582.388} C_VEL
LIN {X 0,Y 677.385,Z 451.058,A -85,B 0,C 180,E1 -4582.648,E2 -4582.648} C_VEL
LIN {X 0,Y 677.229,Z 464.642,A -85,B 0,C 180,E1 -4583.02,E2 -4583.02} C_VEL
LIN {X 0,Y 677.062,Z 478.681,A -85,B 0,C 180,E1 -4583.545,E2 -4583.545} C_VEL
LIN {X 0,Y 676.838,Z 491.017,A -85,B 0,C 180,E1 -4584.135,E2 -4584.135} C_VEL
LIN {X 0,Y 676.666,Z 502.332,A -85,B 0,C 180,E1 -4584.803,E2 -4584.803} C_VEL
LIN {X 0,Y 676.401,Z 512.73,A -85,B 0,C 180,E1 -4585.546,E2 -4585.546} C_VEL
LIN {X 0,Y 676.253,Z 521.443,A -85,B 0,C 180,E1 -4586.288,E2 -4586.288} C_VEL
LIN {X 0,Y 676.042,Z 530.245,A -85,B 0,C 180,E1 -4587.179,E2 -4587.179} C_VEL
LIN {X 0,Y 675.88,Z 537.584,A -85,B 0,C 180,E1 -4588.07,E2 -4588.07} C_VEL
LIN {X 0,Y 675.754,Z 544.619,A -85,B 0,C 180,E1 -4589.109,E2 -4589.109} C_VEL
LIN {X 0,Y 675.629,Z 550.942,A -85,B 0,C 180,E1 -4590.297,E2 -4590.297} C_VEL
LIN {X 0,Y 675.529,Z 554.639,A -85,B 0,C 180,E1 -4591.188,E2 -4591.188} C_VEL
LIN {X 0,Y 675.522,Z 558.256,A -85,B 0,C 180,E1 -4592.377,E2 -4592.377} C_VEL
LIN {X 0,Y 675.519,Z 560.513,A -85,B 0,C 180,E1 -4593.567,E2 -4593.567} C_VEL
LIN {X 0,Y 675.489,Z 561.469,A -85,B 0,C 180,E1 -4594.759,E2 -4594.759} C_VEL
LIN {X 0,Y 675.53,Z 561.125,A -85,B 0,C 180,E1 -4595.952,E2 -4595.952} C_VEL
LIN {X 0,Y 675.557,Z 559.474,A -85,B 0,C 180,E1 -4597.147,E2 -4597.147} C_VEL
LIN {X 0,Y 675.532,Z 558.197,A -85,B 0,C 180,E1 -4597.747,E2 -4597.747} C_VEL
LIN {X 0,Y 675.62,Z 554.485,A -85,B 0,C 180,E1 -4598.947,E2 -4598.947} C_VEL
LIN {X 0,Y 675.705,Z 549.954,A -85,B 0,C 180,E1 -4600.006,E2 -4600.006} C_VEL
LIN {X 0,Y 675.783,Z 544.197,A -85,B 0,C 180,E1 -4601.055,E2 -4601.055} C_VEL
LIN {X 0,Y 675.927,Z 538.065,A -85,B 0,C 180,E1 -4601.962,E2 -4601.962} C_VEL
LIN {X 0,Y 676.085,Z 531.156,A -85,B 0,C 180,E1 -4602.813,E2 -4602.813} C_VEL
LIN {X 0,Y 676.207,Z 523.332,A -85,B 0,C 180,E1 -4603.63,E2 -4603.63} C_VEL
LIN {X 0,Y 676.401,Z 514.729,A -85,B 0,C 180,E1 -4604.391,E2 -4604.391} C_VEL
LIN {X 0,Y 676.592,Z 504.439,A -85,B 0,C 180,E1 -4605.153,E2 -4605.153} C_VEL
LIN {X 0,Y 676.824,Z 493.88,A -85,B 0,C 180,E1 -4605.803,E2 -4605.803} C_VEL
LIN {X 0,Y 677.041,Z 480.924,A -85,B 0,C 180,E1 -4606.452,E2 -4606.452} C_VEL
LIN {X 0,Y 677.208,Z 467.111,A -85,B 0,C 180,E1 -4606.989,E2 -4606.989} C_VEL
LIN {X 0,Y 677.317,Z 452.409,A -85,B 0,C 180,E1 -4607.413,E2 -4607.413} C_VEL
LIN {X 0,Y 677.443,Z 438.339,A -85,B 0,C 180,E1 -4607.686,E2 -4607.686} C_VEL
LIN {X 0,Y 677.701,Z 319.496,A -85,B 0,C 180,E1 -4608.97,E2 -4608.97} C_VEL
LIN {X 0,Y 675.963,Z 313.842,A -85,B 0,C 180,E1 -4609.081,E2 -4609.081} C_VEL
LIN {X 0,Y 675.932,Z 313.846,A -85,B 0,C 180,E1 -4611.904,E2 -4611.904} C_VEL
LIN {X 0,Y 675.914,Z 313.854,A -85,B 0,C 180,E1 -4614.489,E2 -4614.489} C_VEL
LIN {X 0,Y 675.91,Z 313.845,A -85,B 0,C 180,E1 -4617.128,E2 -4617.128} C_VEL
LIN {X 0,Y 675.942,Z 313.839,A -85,B 0,C 180,E1 -4619.488,E2 -4619.488} C_VEL
LIN {X 0,Y 675.904,Z 313.847,A -85,B 0,C 180,E1 -4621.906,E2 -4621.906} C_VEL
LIN {X 0,Y 675.895,Z 313.851,A -85,B 0,C 180,E1 -4624.029,E2 -4624.029} C_VEL
LIN {X 0,Y 675.913,Z 313.852,A -85,B 0,C 180,E1 -4626.206,E2 -4626.206} C_VEL
LIN {X 0,Y 675.922,Z 313.848,A -85,B 0,C 180,E1 -4628.446,E2 -4628.446} C_VEL
LIN {X 0,Y 675.912,Z 313.844,A -85,B 0,C 180,E1 -4630.843,E2 -4630.843} C_VEL
LIN {X 0,Y 675.913,Z 313.844,A -85,B 0,C 180,E1 -4633.497,E2 -4633.497} C_VEL
LIN {X 0,Y 675.943,Z 313.849,A -85,B 0,C 180,E1 -4636.029,E2 -4636.029} C_VEL
LIN {X 0,Y 675.917,Z 313.845,A -85,B 0,C 180,E1 -4638.453,E2 -4638.453} C_VEL
LIN {X 0,Y 675.912,Z 313.84,A -85,B 0,C 180,E1 -4641.007,E2 -4641.007} C_VEL
LIN {X 0,Y 675.908,Z 313.834,A -85,B 0,C 180,E1 -4643.054,E2 -4643.054} C_VEL
LIN {X 0,Y 675.914,Z 313.839,A -85,B 0,C 180,E1 -4645.252,E2 -4645.252} C_VEL
LIN {X 0,Y 675.936,Z 313.842,A -85,B 0,C 180,E1 -4647.394,E2 -4647.394} C_VEL
LIN {X 0,Y 675.917,Z 313.844,A -85,B 0,C 180,E1 -4649.484,E2 -4649.484} C_VEL
LIN {X 0,Y 675.926,Z 313.85,A -85,B 0,C 180,E1 -4651.744,E2 -4651.744} C_VEL
LIN {X 0,Y 675.922,Z 313.84,A -85,B 0,C 180,E1 -4654.365,E2 -4654.365} C_VEL
LIN {X 0,Y 675.916,Z 313.841,A -85,B 0,C 180,E1 -4656.809,E2 -4656.809} C_VEL
LIN {X 0,Y 675.903,Z 313.847,A -85,B 0,C 180,E1 -4659.369,E2 -4659.369} C_VEL
LIN {X 0,Y 675.949,Z 313.847,A -85,B 0,C 180,E1 -4661.888,E2 -4661.888} C_VEL
LIN {X 0,Y 675.955,Z 313.84,A -85,B 0,C 180,E1 -4664.515,E2 -4664.515} C_VEL
LIN {X 0,Y 675.965,Z 313.842,A -85,B 0,C 180,E1 -4665.063,E2 -4665.063} C_VEL
LIN {X 0,Y 677.502,Z 318.894,A -85,B 0,C 180,E1 -4665.159,E2 -4665.159} C_VEL
LIN {X 0,Y 677.281,Z 436.696,A -85,B 0,C 180,E1 -4666.463,E2 -4666.463} C_VEL
LIN {X 0,Y 677.103,Z 450.832,A -85,B 0,C 180,E1 -4666.739,E2 -4666.739} C_VEL
LIN {X 0,Y 676.967,Z 463.94,A -85,B 0,C 180,E1 -4667.108,E2 -4667.108} C_VEL
LIN {X 0,Y 676.82,Z 477.065,A -85,B 0,C 180,E1 -4667.599,E2 -4667.599} C_VEL
LIN {X 0,Y 676.62,Z 488.286,A -85,B 0,C 180,E1 -4668.127,E2 -4668.127} C_VEL
LIN {X 0,Y 676.389,Z 500.065,A -85,B 0,C 180,E1 -4668.804,E2 -4668.804} C_VEL
LIN {X 0,Y 676.216,Z 510.811,A -85,B 0,C 180,E1 -4669.556,E2 -4669.556} C_VEL
LIN {X 0,Y 676.04,Z 521.393,A -85,B 0,C 180,E1 -4670.458,E2 -4670.458} C_VEL
LIN {X 0,Y 675.854,Z 530.085,A -85,B 0,C 180,E1 -4671.357,E2 -4671.357} C_VEL
LIN {X 0,Y 675.693,Z 538.382,A -85,B 0,C 180,E1 -4672.405,E2 -4672.405} C_VEL
LIN {X 0,Y 675.573,Z 545.047,A -85,B 0,C 180,E1 -4673.451,E2 -4673.451} C_VEL
LIN {X 0,Y 675.507,Z 549.778,A -85,B 0,C 180,E1 -4674.376,E2 -4674.376} C_VEL
LIN {X 0,Y 675.525,Z 553.361,A -85,B 0,C 180,E1 -4675.242,E2 -4675.242} C_VEL
LIN {X 0,Y 675.438,Z 555.401,A -85,B 0,C 180,E1 -4675.837,E2 -4675.837} C_VEL
LIN {X 0,Y 675.474,Z 558.307,A -85,B 0,C 180,E1 -4677.028,E2 -4677.028} C_VEL
LIN {X 0,Y 675.41,Z 559.885,A -85,B 0,C 180,E1 -4678.217,E2 -4678.217} C_VEL
LIN {X 0,Y 675.36,Z 560.148,A -85,B 0,C 180,E1 -4679.406,E2 -4679.406} C_VEL
LIN {X 0,Y 675.364,Z 559.115,A -85,B 0,C 180,E1 -4680.594,E2 -4680.594} C_VEL
LIN {X 0,Y 675.389,Z 558.161,A -85,B 0,C 180,E1 -4681.188,E2 -4681.188} C_VEL
LIN {X 0,Y 675.498,Z 555.103,A -85,B 0,C 180,E1 -4682.377,E2 -4682.377} C_VEL
LIN {X 0,Y 675.53,Z 551.921,A -85,B 0,C 180,E1 -4683.269,E2 -4683.269} C_VEL
LIN {X 0,Y 675.577,Z 546.257,A -85,B 0,C 180,E1 -4684.46,E2 -4684.46} C_VEL
LIN {X 0,Y 675.736,Z 540.897,A -85,B 0,C 180,E1 -4685.353,E2 -4685.353} C_VEL
LIN {X 0,Y 675.833,Z 534.413,A -85,B 0,C 180,E1 -4686.247,E2 -4686.247} C_VEL
LIN {X 0,Y 675.951,Z 526.605,A -85,B 0,C 180,E1 -4687.143,E2 -4687.143} C_VEL
LIN {X 0,Y 676.147,Z 517.178,A -85,B 0,C 180,E1 -4688.039,E2 -4688.039} C_VEL
LIN {X 0,Y 676.315,Z 506.734,A -85,B 0,C 180,E1 -4688.862,E2 -4688.862} C_VEL
LIN {X 0,Y 676.541,Z 495.09,A -85,B 0,C 180,E1 -4689.61,E2 -4689.61} C_VEL
LIN {X 0,Y 676.824,Z 481.71,A -85,B 0,C 180,E1 -4690.301,E2 -4690.301} C_VEL
LIN {X 0,Y 676.942,Z 469.251,A -85,B 0,C 180,E1 -4690.809,E2 -4690.809} C_VEL
LIN {X 0,Y 677.064,Z 455.355,A -85,B 0,C 180,E1 -4691.241,E2 -4691.241} C_VEL
LIN {X 0,Y 677.197,Z 441.569,A -85,B 0,C 180,E1 -4691.541,E2 -4691.541} C_VEL
LIN {X 0,Y 677.252,Z 424.423,A -85,B 0,C 180,E1 -4691.767,E2 -4691.767} C_VEL
LIN {X 0,Y 677.666,Z 319.188,A -85,B 0,C 180,E1 -4692.927,E2 -4692.927} C_VEL
LIN {X 0,Y 676.013,Z 313.836,A -85,B 0,C 180,E1 -4693.038,E2 -4693.038} C_VEL
LIN {X 0,Y 676.007,Z 313.833,A -85,B 0,C 180,E1 -4695.628,E2 -4695.628} C_VEL
LIN {X 0,Y 675.972,Z 313.846,A -85,B 0,C 180,E1 -4698.111,E2 -4698.111} C_VEL
LIN {X 0,Y 675.938,Z 313.844,A -85,B 0,C 180,E1 -4700.63,E2 -4700.63} C_VEL
LIN {X 0,Y 675.959,Z 313.839,A -85,B 0,C 180,E1 -4703.189,E2 -4703.189} C_VEL
LIN {X 0,Y 675.936,Z 313.85,A -85,B 0,C 180,E1 -4705.8,E2 -4705.8} C_VEL
LIN {X 0,Y 675.965,Z 313.84,A -85,B 0,C 180,E1 -4708.263,E2 -4708.263} C_VEL
LIN {X 0,Y 675.99,Z 313.833,A -85,B 0,C 180,E1 -4710.68,E2 -4710.68} C_VEL
LIN {X 0,Y 675.951,Z 313.843,A -85,B 0,C 180,E1 -4713.312,E2 -4713.312} C_VEL
LIN {X 0,Y 675.951,Z 313.846,A -85,B 0,C 180,E1 -4715.471,E2 -4715.471} C_VEL
LIN {X 0,Y 675.941,Z 313.839,A -85,B 0,C 180,E1 -4718.042,E2 -4718.042} C_VEL
LIN {X 0,Y 675.934,Z 313.841,A -85,B 0,C 180,E1 -4720.846,E2 -4720.846} C_VEL
LIN {X 0,Y 675.947,Z 313.842,A -85,B 0,C 180,E1 -4723.5,E2 -4723.5} C_VEL
LIN {X 0,Y 675.941,Z 313.838,A -85,B 0,C 180,E1 -4726.029,E2 -4726.029} C_VEL
LIN {X 0,Y 675.915,Z 313.844,A -85,B 0,C 180,E1 -4728.453,E2 -4728.453} C_VEL
LIN {X 0,Y 675.931,Z 313.848,A -85,B 0,C 180,E1 -4731.005,E2 -4731.005} C_VEL
LIN {X 0,Y 675.91,Z 313.849,A -85,B 0,C 180,E1 -4733.054,E2 -4733.054} C_VEL
LIN {X 0,Y 675.909,Z 313.843,A -85,B 0,C 180,E1 -4735.252,E2 -4735.252} C_VEL
LIN {X 0,Y 675.913,Z 313.844,A -85,B 0,C 180,E1 -4737.393,E2 -4737.393} C_VEL
LIN {X 0,Y 675.913,Z 313.843,A -85,B 0,C 180,E1 -4739.483,E2 -4739.483} C_VEL
LIN {X 0,Y 675.923,Z 313.845,A -85,B 0,C 180,E1 -4741.743,E2 -4741.743} C_VEL
LIN {X 0,Y 675.92,Z 313.928,A -85,B 0,C 180,E1 -4743.849,E2 -4743.849} C_VEL
LIN {X 0,Y 677.734,Z 322.853,A -85,B 0,C 180,E1 -4744.765,E2 -4744.765} C_VEL
LIN {X 0,Y 677.767,Z 331.389,A -85,B 0,C 180,E1 -4745.582,E2 -4745.582} C_VEL
LIN {X 0,Y 677.487,Z 353.543,A -85,B 0,C 180,E1 -4747.669,E2 -4747.669} C_VEL
LIN {X 0,Y 677.1,Z 380.835,A -85,B 0,C 180,E1 -4750.205,E2 -4750.205} C_VEL
LIN {X 0,Y 676.715,Z 407.813,A -85,B 0,C 180,E1 -4752.687,E2 -4752.687} C_VEL
LIN {X 0,Y 676.439,Z 436.472,A -85,B 0,C 180,E1 -4755.304,E2 -4755.304} C_VEL
LIN {X 0,Y 676.347,Z 442.135,A -85,B 0,C 180,E1 -4755.819,E2 -4755.819} C_VEL
LIN {X 0,Y 677.688,Z 455.452,A -85,B 0,C 180,E1 -4756,E2 -4756} C_VEL
LIN {X 0,Y 677.233,Z 581.124,A -85,B 0,C 180,E1 -4757.342,E2 -4757.342} C_VEL
LIN {X 0,Y 677.047,Z 595.219,A -85,B 0,C 180,E1 -4757.604,E2 -4757.604} C_VEL
LIN {X 0,Y 676.889,Z 608.96,A -85,B 0,C 180,E1 -4757.98,E2 -4757.98} C_VEL
LIN {X 0,Y 676.693,Z 621.443,A -85,B 0,C 180,E1 -4758.431,E2 -4758.431} C_VEL
LIN {X 0,Y 676.436,Z 633.073,A -85,B 0,C 180,E1 -4758.956,E2 -4758.956} C_VEL
LIN {X 0,Y 676.244,Z 645.666,A -85,B 0,C 180,E1 -4759.661,E2 -4759.661} C_VEL
LIN {X 0,Y 676.035,Z 657.276,A -85,B 0,C 180,E1 -4760.457,E2 -4760.457} C_VEL
LIN {X 0,Y 675.827,Z 668.068,A -85,B 0,C 180,E1 -4761.357,E2 -4761.357} C_VEL
LIN {X 0,Y 675.71,Z 676.998,A -85,B 0,C 180,E1 -4762.255,E2 -4762.255} C_VEL
LIN {X 0,Y 675.558,Z 685.579,A -85,B 0,C 180,E1 -4763.301,E2 -4763.301} C_VEL
LIN {X 0,Y 675.472,Z 692.492,A -85,B 0,C 180,E1 -4764.347,E2 -4764.347} C_VEL
LIN {X 0,Y 675.438,Z 698.677,A -85,B 0,C 180,E1 -4765.539,E2 -4765.539} C_VEL
LIN {X 0,Y 675.371,Z 702.218,A -85,B 0,C 180,E1 -4766.432,E2 -4766.432} C_VEL
LIN {X 0,Y 675.374,Z 705.669,A -85,B 0,C 180,E1 -4767.622,E2 -4767.622} C_VEL
LIN {X 0,Y 675.336,Z 707.701,A -85,B 0,C 180,E1 -4768.811,E2 -4768.811} C_VEL
LIN {X 0,Y 675.298,Z 708.371,A -85,B 0,C 180,E1 -4770,E2 -4770} C_VEL
LIN {X 0,Y 675.336,Z 707.7,A -85,B 0,C 180,E1 -4771.189,E2 -4771.189} C_VEL
LIN {X 0,Y 675.374,Z 705.665,A -85,B 0,C 180,E1 -4772.378,E2 -4772.378} C_VEL
LIN {X 0,Y 675.371,Z 702.22,A -85,B 0,C 180,E1 -4773.568,E2 -4773.568} C_VEL
LIN {X 0,Y 675.451,Z 697.269,A -85,B 0,C 180,E1 -4774.759,E2 -4774.759} C_VEL
LIN {X 0,Y 675.48,Z 692.505,A -85,B 0,C 180,E1 -4775.653,E2 -4775.653} C_VEL
LIN {X 0,Y 675.558,Z 685.562,A -85,B 0,C 180,E1 -4776.698,E2 -4776.698} C_VEL
LIN {X 0,Y 675.71,Z 677.001,A -85,B 0,C 180,E1 -4777.745,E2 -4777.745} C_VEL
LIN {X 0,Y 675.827,Z 668.084,A -85,B 0,C 180,E1 -4778.643,E2 -4778.643} C_VEL
LIN {X 0,Y 676.036,Z 657.297,A -85,B 0,C 180,E1 -4779.542,E2 -4779.542} C_VEL
LIN {X 0,Y 676.251,Z 645.718,A -85,B 0,C 180,E1 -4780.337,E2 -4780.337} C_VEL
LIN {X 0,Y 676.434,Z 633.099,A -85,B 0,C 180,E1 -4781.044,E2 -4781.044} C_VEL
LIN {X 0,Y 676.71,Z 619.606,A -85,B 0,C 180,E1 -4781.644,E2 -4781.644} C_VEL
LIN {X 0,Y 676.92,Z 606.586,A -85,B 0,C 180,E1 -4782.095,E2 -4782.095} C_VEL
LIN {X 0,Y 677.121,Z 592.645,A -85,B 0,C 180,E1 -4782.452,E2 -4782.452} C_VEL
LIN {X 0,Y 677.254,Z 578.198,A -85,B 0,C 180,E1 -4782.696,E2 -4782.696} C_VEL
LIN {X 0,Y 677.669,Z 453.721,A -85,B 0,C 180,E1 -4784.019,E2 -4784.019} C_VEL
LIN {X 0,Y 676.347,Z 442.177,A -85,B 0,C 180,E1 -4784.181,E2 -4784.181} C_VEL
LIN {X 0,Y 676.698,Z 412.935,A -85,B 0,C 180,E1 -4786.847,E2 -4786.847} C_VEL
LIN {X 0,Y 677.078,Z 383.858,A -85,B 0,C 180,E1 -4789.522,E2 -4789.522} C_VEL
LIN {X 0,Y 677.42,Z 358.75,A -85,B 0,C 180,E1 -4791.854,E2 -4791.854} C_VEL
LIN {X 0,Y 677.746,Z 334.867,A -85,B 0,C 180,E1 -4794.094,E2 -4794.094} C_VEL
LIN {X 0,Y 677.731,Z 322.843,A -85,B 0,C 180,E1 -4795.235,E2 -4795.235} C_VEL
LIN {X 0,Y 675.931,Z 313.849,A -85,B 0,C 180,E1 -4796.171,E2 -4796.171} C_VEL
LIN {X 0,Y 675.917,Z 313.844,A -85,B 0,C 180,E1 -4798.47,E2 -4798.47} C_VEL
LIN {X 0,Y 675.924,Z 313.841,A -85,B 0,C 180,E1 -4800.671,E2 -4800.671} C_VEL
LIN {X 0,Y 675.918,Z 313.85,A -85,B 0,C 180,E1 -4803.314,E2 -4803.314} C_VEL
LIN {X 0,Y 675.913,Z 313.844,A -85,B 0,C 180,E1 -4806.069,E2 -4806.069} C_VEL
LIN {X 0,Y 675.906,Z 313.844,A -85,B 0,C 180,E1 -4808.446,E2 -4808.446} C_VEL
LIN {X 0,Y 675.907,Z 313.848,A -85,B 0,C 180,E1 -4810.843,E2 -4810.843} C_VEL
LIN {X 0,Y 675.909,Z 313.85,A -85,B 0,C 180,E1 -4813.497,E2 -4813.497} C_VEL
LIN {X 0,Y 675.934,Z 313.841,A -85,B 0,C 180,E1 -4816.029,E2 -4816.029} C_VEL
LIN {X 0,Y 675.913,Z 313.846,A -85,B 0,C 180,E1 -4818.454,E2 -4818.454} C_VEL
LIN {X 0,Y 675.912,Z 313.853,A -85,B 0,C 180,E1 -4821.007,E2 -4821.007} C_VEL
LIN {X 0,Y 675.91,Z 313.851,A -85,B 0,C 180,E1 -4823.055,E2 -4823.055} C_VEL
LIN {X 0,Y 675.932,Z 313.845,A -85,B 0,C 180,E1 -4825.254,E2 -4825.254} C_VEL
LIN {X 0,Y 675.933,Z 313.845,A -85,B 0,C 180,E1 -4827.394,E2 -4827.394} C_VEL
LIN {X 0,Y 675.918,Z 313.848,A -85,B 0,C 180,E1 -4829.484,E2 -4829.484} C_VEL
LIN {X 0,Y 675.924,Z 313.847,A -85,B 0,C 180,E1 -4831.743,E2 -4831.743} C_VEL
LIN {X 0,Y 675.984,Z 313.979,A -85,B 0,C 180,E1 -4834.299,E2 -4834.299} C_VEL
LIN {X 0,Y 677.704,Z 323.695,A -85,B 0,C 180,E1 -4835.227,E2 -4835.227} C_VEL
LIN {X 0,Y 677.568,Z 350.606,A -85,B 0,C 180,E1 -4837.672,E2 -4837.672} C_VEL
LIN {X 0,Y 677.303,Z 379.619,A -85,B 0,C 180,E1 -4840.332,E2 -4840.332} C_VEL
LIN {X 0,Y 676.93,Z 405.308,A -85,B 0,C 180,E1 -4842.693,E2 -4842.693} C_VEL
LIN {X 0,Y 676.663,Z 428.296,A -85,B 0,C 180,E1 -4844.848,E2 -4844.848} C_VEL
LIN {X 0,Y 676.544,Z 439.644,A -85,B 0,C 180,E1 -4845.89,E2 -4845.89} C_VEL
LIN {X 0,Y 677.685,Z 448.934,A -85,B 0,C 180,E1 -4846.019,E2 -4846.019} C_VEL
LIN {X 0,Y 677.226,Z 578.289,A -85,B 0,C 180,E1 -4847.437,E2 -4847.437} C_VEL
LIN {X 0,Y 677.045,Z 592.169,A -85,B 0,C 180,E1 -4847.699,E2 -4847.699} C_VEL
LIN {X 0,Y 676.884,Z 605.328,A -85,B 0,C 180,E1 -4848.056,E2 -4848.056} C_VEL
LIN {X 0,Y 676.646,Z 619.658,A -85,B 0,C 180,E1 -4848.581,E2 -4848.581} C_VEL
LIN {X 0,Y 676.405,Z 630.872,A -85,B 0,C 180,E1 -4849.106,E2 -4849.106} C_VEL
LIN {X 0,Y 676.273,Z 641.702,A -85,B 0,C 180,E1 -4849.723,E2 -4849.723} C_VEL
LIN {X 0,Y 676.117,Z 651.434,A -85,B 0,C 180,E1 -4850.384,E2 -4850.384} C_VEL
LIN {X 0,Y 675.929,Z 659.9,A -85,B 0,C 180,E1 -4851.058,E2 -4851.058} C_VEL
LIN {X 0,Y 675.757,Z 669.464,A -85,B 0,C 180,E1 -4851.956,E2 -4851.956} C_VEL
LIN {X 0,Y 675.632,Z 678.527,A -85,B 0,C 180,E1 -4853.003,E2 -4853.003} C_VEL
LIN {X 0,Y 675.554,Z 683.936,A -85,B 0,C 180,E1 -4853.75,E2 -4853.75} C_VEL
LIN {X 0,Y 675.442,Z 690.145,A -85,B 0,C 180,E1 -4854.799,E2 -4854.799} C_VEL
LIN {X 0,Y 675.394,Z 695.006,A -85,B 0,C 180,E1 -4855.837,E2 -4855.837} C_VEL
LIN {X 0,Y 675.372,Z 697.332,A -85,B 0,C 180,E1 -4856.432,E2 -4856.432} C_VEL
LIN {X 0,Y 675.374,Z 700.724,A -85,B 0,C 180,E1 -4857.623,E2 -4857.623} C_VEL
LIN {X 0,Y 675.34,Z 702.77,A -85,B 0,C 180,E1 -4858.812,E2 -4858.812} C_VEL
LIN {X 0,Y 675.297,Z 703.501,A -85,B 0,C 180,E1 -4860,E2 -4860} C_VEL
LIN {X 0,Y 675.338,Z 702.856,A -85,B 0,C 180,E1 -4861.189,E2 -4861.189} C_VEL
LIN {X 0,Y 675.373,Z 700.928,A -85,B 0,C 180,E1 -4862.378,E2 -4862.378} C_VEL
LIN {X 0,Y 675.417,Z 699.469,A -85,B 0,C 180,E1 -4862.972,E2 -4862.972} C_VEL
LIN {X 0,Y 675.394,Z 695.375,A -85,B 0,C 180,E1 -4864.163,E2 -4864.163} C_VEL
LIN {X 0,Y 675.462,Z 691.738,A -85,B 0,C 180,E1 -4864.98,E2 -4864.98} C_VEL
LIN {X 0,Y 675.487,Z 686.353,A -85,B 0,C 180,E1 -4865.952,E2 -4865.952} C_VEL
LIN {X 0,Y 675.575,Z 680.295,A -85,B 0,C 180,E1 -4866.848,E2 -4866.848} C_VEL
LIN {X 0,Y 675.687,Z 673.035,A -85,B 0,C 180,E1 -4867.745,E2 -4867.745} C_VEL
LIN {X 0,Y 675.859,Z 664.342,A -85,B 0,C 180,E1 -4868.643,E2 -4868.643} C_VEL
LIN {X 0,Y 676.072,Z 653.728,A -85,B 0,C 180,E1 -4869.542,E2 -4869.542} C_VEL
LIN {X 0,Y 676.246,Z 643.409,A -85,B 0,C 180,E1 -4870.264,E2 -4870.264} C_VEL
LIN {X 0,Y 676.409,Z 632.646,A -85,B 0,C 180,E1 -4870.894,E2 -4870.894} C_VEL
LIN {X 0,Y 676.65,Z 621.819,A -85,B 0,C 180,E1 -4871.419,E2 -4871.419} C_VEL
LIN {X 0,Y 676.887,Z 608.362,A -85,B 0,C 180,E1 -4871.944,E2 -4871.944} C_VEL
LIN {X 0,Y 677.042,Z 594.009,A -85,B 0,C 180,E1 -4872.359,E2 -4872.359} C_VEL
LIN {X 0,Y 677.172,Z 580.943,A -85,B 0,C 180,E1 -4872.622,E2 -4872.622} C_VEL
LIN {X 0,Y 677.3,Z 562.841,A -85,B 0,C 180,E1 -4872.847,E2 -4872.847} C_VEL
LIN {X 0,Y 677.583,Z 447.46,A -85,B 0,C 180,E1 -4874.091,E2 -4874.091} C_VEL
LIN {X 0,Y 676.525,Z 439.533,A -85,B 0,C 180,E1 -4874.216,E2 -4874.216} C_VEL
LIN {X 0,Y 676.873,Z 414.832,A -85,B 0,C 180,E1 -4876.534,E2 -4876.534} C_VEL
LIN {X 0,Y 677.318,Z 386.845,A -85,B 0,C 180,E1 -4879.168,E2 -4879.168} C_VEL
LIN {X 0,Y 677.651,Z 365.22,A -85,B 0,C 180,E1 -4881.209,E2 -4881.209} C_VEL
LIN {X 0,Y 677.082,Z 361.396,A -85,B 0,C 180,E1 -4881.586,E2 -4881.586} C_VEL
LIN {X 0,Y 671.667,Z 349.67,A -85,B 0,C 180,E1 -4882.868,E2 -4882.868} C_VEL
LIN {X 0,Y 671.064,Z 345.871,A -85,B 0,C 180,E1 -4883.252,E2 -4883.252} C_VEL
LIN {X 0,Y 671.328,Z 326.035,A -85,B 0,C 180,E1 -4885.156,E2 -4885.156} C_VEL
LIN {X 0,Y 668.905,Z 314.722,A -85,B 0,C 180,E1 -4886.342,E2 -4886.342} C_VEL
LIN {X 0,Y 668.918,Z 314.718,A -85,B 0,C 180,E1 -4888.795,E2 -4888.795} C_VEL
LIN {X 0,Y 668.934,Z 314.715,A -85,B 0,C 180,E1 -4890.87,E2 -4890.87} C_VEL
LIN {X 0,Y 668.911,Z 314.718,A -85,B 0,C 180,E1 -4893.71,E2 -4893.71} C_VEL
LIN {X 0,Y 668.895,Z 314.716,A -85,B 0,C 180,E1 -4896.262,E2 -4896.262} C_VEL
LIN {X 0,Y 668.891,Z 314.724,A -85,B 0,C 180,E1 -4898.925,E2 -4898.925} C_VEL
LIN {X 0,Y 668.916,Z 314.72,A -85,B 0,C 180,E1 -4901.277,E2 -4901.277} C_VEL
LIN {X 0,Y 668.93,Z 314.712,A -85,B 0,C 180,E1 -4903.738,E2 -4903.738} C_VEL
LIN {X 0,Y 668.936,Z 314.714,A -85,B 0,C 180,E1 -4906.284,E2 -4906.284} C_VEL
LIN {X 0,Y 668.919,Z 314.721,A -85,B 0,C 180,E1 -4908.933,E2 -4908.933} C_VEL
LIN {X 0,Y 668.896,Z 314.72,A -85,B 0,C 180,E1 -4911.075,E2 -4911.075} C_VEL
LIN {X 0,Y 668.896,Z 314.717,A -85,B 0,C 180,E1 -4913.738,E2 -4913.738} C_VEL
LIN {X 0,Y 668.912,Z 314.721,A -85,B 0,C 180,E1 -4916.29,E2 -4916.29} C_VEL
LIN {X 0,Y 668.919,Z 314.714,A -85,B 0,C 180,E1 -4919.165,E2 -4919.165} C_VEL
LIN {X 0,Y 668.917,Z 314.715,A -85,B 0,C 180,E1 -4921.594,E2 -4921.594} C_VEL
LIN {X 0,Y 668.9,Z 314.727,A -85,B 0,C 180,E1 -4924.232,E2 -4924.232} C_VEL
LIN {X 0,Y 668.943,Z 314.711,A -85,B 0,C 180,E1 -4927.206,E2 -4927.206} C_VEL
LIN {X 0,Y 668.899,Z 314.723,A -85,B 0,C 180,E1 -4929.784,E2 -4929.784} C_VEL
LIN {X 0,Y 668.949,Z 314.714,A -85,B 0,C 180,E1 -4932.336,E2 -4932.336} C_VEL
LIN {X 0,Y 668.922,Z 314.713,A -85,B 0,C 180,E1 -4934.824,E2 -4934.824} C_VEL
LIN {X 0,Y 668.954,Z 314.713,A -85,B 0,C 180,E1 -4937.298,E2 -4937.298} C_VEL
LIN {X 0,Y 668.991,Z 314.706,A -85,B 0,C 180,E1 -4940.356,E2 -4940.356} C_VEL
LIN {X 0,Y 668.953,Z 314.897,A -85,B 0,C 180,E1 -4940.875,E2 -4940.875} C_VEL
LIN {X 0,Y 670.924,Z 321.462,A -85,B 0,C 180,E1 -4940.99,E2 -4940.99} C_VEL
LIN {X 0,Y 670.575,Z 437.649,A -85,B 0,C 180,E1 -4942.252,E2 -4942.252} C_VEL
LIN {X 0,Y 670.511,Z 451.711,A -85,B 0,C 180,E1 -4942.516,E2 -4942.516} C_VEL
LIN {X 0,Y 670.323,Z 465.845,A -85,B 0,C 180,E1 -4942.91,E2 -4942.91} C_VEL
LIN {X 0,Y 670.174,Z 478.823,A -85,B 0,C 180,E1 -4943.398,E2 -4943.398} C_VEL
LIN {X 0,Y 669.939,Z 491.358,A -85,B 0,C 180,E1 -4943.999,E2 -4943.999} C_VEL
LIN {X 0,Y 669.714,Z 503.899,A -85,B 0,C 180,E1 -4944.749,E2 -4944.749} C_VEL
LIN {X 0,Y 669.444,Z 514.165,A -85,B 0,C 180,E1 -4945.499,E2 -4945.499} C_VEL
LIN {X 0,Y 669.183,Z 524.368,A -85,B 0,C 180,E1 -4946.399,E2 -4946.399} C_VEL
LIN {X 0,Y 668.979,Z 532.807,A -85,B 0,C 180,E1 -4947.3,E2 -4947.3} C_VEL
LIN {X 0,Y 668.871,Z 540.911,A -85,B 0,C 180,E1 -4948.35,E2 -4948.35} C_VEL
LIN {X 0,Y 668.675,Z 547.45,A -85,B 0,C 180,E1 -4949.4,E2 -4949.4} C_VEL
LIN {X 0,Y 668.53,Z 553.25,A -85,B 0,C 180,E1 -4950.6,E2 -4950.6} C_VEL
LIN {X 0,Y 668.443,Z 557.515,A -85,B 0,C 180,E1 -4951.802,E2 -4951.802} C_VEL
LIN {X 0,Y 668.493,Z 560.385,A -85,B 0,C 180,E1 -4953.003,E2 -4953.003} C_VEL
LIN {X 0,Y 668.491,Z 561.943,A -85,B 0,C 180,E1 -4954.206,E2 -4954.206} C_VEL
LIN {X 0,Y 668.439,Z 562.208,A -85,B 0,C 180,E1 -4955.442,E2 -4955.442} C_VEL
LIN {X 0,Y 668.485,Z 561.184,A -85,B 0,C 180,E1 -4956.619,E2 -4956.619} C_VEL
LIN {X 0,Y 668.479,Z 558.836,A -85,B 0,C 180,E1 -4957.829,E2 -4957.829} C_VEL
LIN {X 0,Y 668.607,Z 555.056,A -85,B 0,C 180,E1 -4959.041,E2 -4959.041} C_VEL
LIN {X 0,Y 668.678,Z 550.785,A -85,B 0,C 180,E1 -4960.048,E2 -4960.048} C_VEL
LIN {X 0,Y 668.793,Z 544.65,A -85,B 0,C 180,E1 -4961.172,E2 -4961.172} C_VEL
LIN {X 0,Y 668.972,Z 537.311,A -85,B 0,C 180,E1 -4962.241,E2 -4962.241} C_VEL
LIN {X 0,Y 669.157,Z 529.027,A -85,B 0,C 180,E1 -4963.222,E2 -4963.222} C_VEL
LIN {X 0,Y 669.327,Z 520.279,A -85,B 0,C 180,E1 -4964.082,E2 -4964.082} C_VEL
LIN {X 0,Y 669.577,Z 508.812,A -85,B 0,C 180,E1 -4965.006,E2 -4965.006} C_VEL
LIN {X 0,Y 669.823,Z 497.053,A -85,B 0,C 180,E1 -4965.777,E2 -4965.777} C_VEL
LIN {X 0,Y 670.058,Z 485.48,A -85,B 0,C 180,E1 -4966.394,E2 -4966.394} C_VEL
LIN {X 0,Y 670.26,Z 471.819,A -85,B 0,C 180,E1 -4966.975,E2 -4966.975} C_VEL
LIN {X 0,Y 670.434,Z 458.613,A -85,B 0,C 180,E1 -4967.402,E2 -4967.402} C_VEL
LIN {X 0,Y 670.503,Z 444.556,A -85,B 0,C 180,E1 -4967.727,E2 -4967.727} C_VEL
LIN {X 0,Y 670.588,Z 428.746,A -85,B 0,C 180,E1 -4967.947,E2 -4967.947} C_VEL
LIN {X 0,Y 670.791,Z 320.598,A -85,B 0,C 180,E1 -4969.114,E2 -4969.114} C_VEL
LIN {X 0,Y 668.918,Z 314.719,A -85,B 0,C 180,E1 -4969.237,E2 -4969.237} C_VEL
LIN {X 0,Y 668.879,Z 314.728,A -85,B 0,C 180,E1 -4972.147,E2 -4972.147} C_VEL
LIN {X 0,Y 668.874,Z 314.728,A -85,B 0,C 180,E1 -4974.764,E2 -4974.764} C_VEL
LIN {X 0,Y 668.855,Z 314.723,A -85,B 0,C 180,E1 -4977.438,E2 -4977.438} C_VEL
LIN {X 0,Y 668.864,Z 314.73,A -85,B 0,C 180,E1 -4980.177,E2 -4980.177} C_VEL
LIN {X 0,Y 668.856,Z 314.732,A -85,B 0,C 180,E1 -4982.282,E2 -4982.282} C_VEL
LIN {X 0,Y 668.879,Z 314.719,A -85,B 0,C 180,E1 -4985.167,E2 -4985.167} C_VEL
LIN {X 0,Y 668.875,Z 314.719,A -85,B 0,C 180,E1 -4987.4,E2 -4987.4} C_VEL
LIN {X 0,Y 668.863,Z 314.731,A -85,B 0,C 180,E1 -4990.14,E2 -4990.14} C_VEL
LIN {X 0,Y 668.863,Z 314.731,A -85,B 0,C 180,E1 -4992.084,E2 -4992.084} C_VEL
LIN {X 0,Y 668.905,Z 314.717,A -85,B 0,C 180,E1 -4994.597,E2 -4994.597} C_VEL
LIN {X 0,Y 668.857,Z 314.721,A -85,B 0,C 180,E1 -4997.144,E2 -4997.144} C_VEL
LIN {X 0,Y 668.865,Z 314.723,A -85,B 0,C 180,E1 -4999.513,E2 -4999.513} C_VEL
LIN {X 0,Y 668.897,Z 314.722,A -85,B 0,C 180,E1 -5001.842,E2 -5001.842} C_VEL
LIN {X 0,Y 668.885,Z 314.721,A -85,B 0,C 180,E1 -5004.096,E2 -5004.096} C_VEL
LIN {X 0,Y 668.898,Z 314.715,A -85,B 0,C 180,E1 -5006.902,E2 -5006.902} C_VEL
LIN {X 0,Y 668.88,Z 314.717,A -85,B 0,C 180,E1 -5009.171,E2 -5009.171} C_VEL
LIN {X 0,Y 668.877,Z 314.725,A -85,B 0,C 180,E1 -5011.6,E2 -5011.6} C_VEL
LIN {X 0,Y 668.884,Z 314.718,A -85,B 0,C 180,E1 -5014.235,E2 -5014.235} C_VEL
LIN {X 0,Y 668.869,Z 314.719,A -85,B 0,C 180,E1 -5016.55,E2 -5016.55} C_VEL
LIN {X 0,Y 668.879,Z 314.719,A -85,B 0,C 180,E1 -5019.142,E2 -5019.142} C_VEL
LIN {X 0,Y 668.89,Z 314.73,A -85,B 0,C 180,E1 -5021.69,E2 -5021.69} C_VEL
LIN {X 0,Y 668.909,Z 314.719,A -85,B 0,C 180,E1 -5024.446,E2 -5024.446} C_VEL
LIN {X 0,Y 668.904,Z 314.721,A -85,B 0,C 180,E1 -5024.921,E2 -5024.921} C_VEL
LIN {X 0,Y 670.728,Z 321.091,A -85,B 0,C 180,E1 -5025.04,E2 -5025.04} C_VEL
LIN {X 0,Y 670.341,Z 437.191,A -85,B 0,C 180,E1 -5026.343,E2 -5026.343} C_VEL
LIN {X 0,Y 670.155,Z 451.799,A -85,B 0,C 180,E1 -5026.631,E2 -5026.631} C_VEL
LIN {X 0,Y 670.021,Z 466.164,A -85,B 0,C 180,E1 -5027.049,E2 -5027.049} C_VEL
LIN {X 0,Y 669.864,Z 478.974,A -85,B 0,C 180,E1 -5027.545,E2 -5027.545} C_VEL
LIN {X 0,Y 669.661,Z 491.429,A -85,B 0,C 180,E1 -5028.154,E2 -5028.154} C_VEL
LIN {X 0,Y 669.406,Z 502.75,A -85,B 0,C 180,E1 -5028.838,E2 -5028.838} C_VEL
LIN {X 0,Y 669.159,Z 514.64,A -85,B 0,C 180,E1 -5029.722,E2 -5029.722} C_VEL
LIN {X 0,Y 669.003,Z 524.948,A -85,B 0,C 180,E1 -5030.66,E2 -5030.66} C_VEL
LIN {X 0,Y 668.823,Z 533.177,A -85,B 0,C 180,E1 -5031.569,E2 -5031.569} C_VEL
LIN {X 0,Y 668.675,Z 541.045,A -85,B 0,C 180,E1 -5032.627,E2 -5032.627} C_VEL
LIN {X 0,Y 668.557,Z 547.358,A -85,B 0,C 180,E1 -5033.684,E2 -5033.684} C_VEL
LIN {X 0,Y 668.469,Z 552.536,A -85,B 0,C 180,E1 -5034.793,E2 -5034.793} C_VEL
LIN {X 0,Y 668.401,Z 556.094,A -85,B 0,C 180,E1 -5035.793,E2 -5035.793} C_VEL
LIN {X 0,Y 668.435,Z 559.029,A -85,B 0,C 180,E1 -5036.996,E2 -5036.996} C_VEL
LIN {X 0,Y 668.351,Z 560.635,A -85,B 0,C 180,E1 -5038.198,E2 -5038.198} C_VEL
LIN {X 0,Y 668.304,Z 560.936,A -85,B 0,C 180,E1 -5039.399,E2 -5039.399} C_VEL
LIN {X 0,Y 668.312,Z 559.927,A -85,B 0,C 180,E1 -5040.6,E2 -5040.6} C_VEL
LIN {X 0,Y 668.386,Z 557.597,A -85,B 0,C 180,E1 -5041.801,E2 -5041.801} C_VEL
LIN {X 0,Y 668.48,Z 553.886,A -85,B 0,C 180,E1 -5043.003,E2 -5043.003} C_VEL
LIN {X 0,Y 668.523,Z 548.637,A -85,B 0,C 180,E1 -5044.206,E2 -5044.206} C_VEL
LIN {X 0,Y 668.728,Z 541.706,A -85,B 0,C 180,E1 -5045.409,E2 -5045.409} C_VEL
LIN {X 0,Y 668.841,Z 534.012,A -85,B 0,C 180,E1 -5046.464,E2 -5046.464} C_VEL
LIN {X 0,Y 669.037,Z 525.946,A -85,B 0,C 180,E1 -5047.368,E2 -5047.368} C_VEL
LIN {X 0,Y 669.2,Z 516.174,A -85,B 0,C 180,E1 -5048.275,E2 -5048.275} C_VEL
LIN {X 0,Y 669.396,Z 505.283,A -85,B 0,C 180,E1 -5049.106,E2 -5049.106} C_VEL
LIN {X 0,Y 669.61,Z 494.463,A -85,B 0,C 180,E1 -5049.787,E2 -5049.787} C_VEL
LIN {X 0,Y 669.893,Z 481.697,A -85,B 0,C 180,E1 -5050.44,E2 -5050.44} C_VEL
LIN {X 0,Y 670.002,Z 468.805,A -85,B 0,C 180,E1 -5050.961,E2 -5050.961} C_VEL
LIN {X 0,Y 670.137,Z 455.052,A -85,B 0,C 180,E1 -5051.378,E2 -5051.378} C_VEL
LIN {X 0,Y 670.265,Z 440.71,A -85,B 0,C 180,E1 -5051.682,E2 -5051.682} C_VEL
LIN {X 0,Y 670.349,Z 419.184,A -85,B 0,C 180,E1 -5051.948,E2 -5051.948} C_VEL
LIN {X 0,Y 670.696,Z 320.364,A -85,B 0,C 180,E1 -5053.06,E2 -5053.06} C_VEL
LIN {X 0,Y 668.95,Z 314.715,A -85,B 0,C 180,E1 -5053.173,E2 -5053.173} C_VEL
LIN {X 0,Y 668.968,Z 314.712,A -85,B 0,C 180,E1 -5055.797,E2 -5055.797} C_VEL
LIN {X 0,Y 668.919,Z 314.725,A -85,B 0,C 180,E1 -5058.309,E2 -5058.309} C_VEL
LIN {X 0,Y 668.92,Z 314.717,A -85,B 0,C 180,E1 -5060.856,E2 -5060.856} C_VEL
LIN {X 0,Y 668.921,Z 314.718,A -85,B 0,C 180,E1 -5063.447,E2 -5063.447} C_VEL
LIN {X 0,Y 668.892,Z 314.727,A -85,B 0,C 180,E1 -5066.092,E2 -5066.092} C_VEL
LIN {X 0,Y 668.918,Z 314.716,A -85,B 0,C 180,E1 -5068.406,E2 -5068.406} C_VEL
LIN {X 0,Y 668.93,Z 314.713,A -85,B 0,C 180,E1 -5070.869,E2 -5070.869} C_VEL
LIN {X 0,Y 668.911,Z 314.723,A -85,B 0,C 180,E1 -5073.71,E2 -5073.71} C_VEL
LIN {X 0,Y 668.894,Z 314.716,A -85,B 0,C 180,E1 -5076.262,E2 -5076.262} C_VEL
LIN {X 0,Y 668.888,Z 314.719,A -85,B 0,C 180,E1 -5078.925,E2 -5078.925} C_VEL
LIN {X 0,Y 668.892,Z 314.725,A -85,B 0,C 180,E1 -5081.278,E2 -5081.278} C_VEL
LIN {X 0,Y 668.897,Z 314.717,A -85,B 0,C 180,E1 -5083.735,E2 -5083.735} C_VEL
LIN {X 0,Y 668.9,Z 314.716,A -85,B 0,C 180,E1 -5086.28,E2 -5086.28} C_VEL
LIN {X 0,Y 668.876,Z 314.73,A -85,B 0,C 180,E1 -5088.936,E2 -5088.936} C_VEL
LIN {X 0,Y 668.884,Z 314.725,A -85,B 0,C 180,E1 -5091.074,E2 -5091.074} C_VEL
LIN {X 0,Y 668.861,Z 314.722,A -85,B 0,C 180,E1 -5093.742,E2 -5093.742} C_VEL
LIN {X 0,Y 668.864,Z 314.724,A -85,B 0,C 180,E1 -5096.287,E2 -5096.287} C_VEL
LIN {X 0,Y 668.857,Z 314.731,A -85,B 0,C 180,E1 -5098.425,E2 -5098.425} C_VEL
LIN {X 0,Y 668.914,Z 314.725,A -85,B 0,C 180,E1 -5100.517,E2 -5100.517} C_VEL
LIN {X 0,Y 668.858,Z 314.727,A -85,B 0,C 180,E1 -5103.236,E2 -5103.236} C_VEL
LIN {X 0,Y 668.907,Z 314.828,A -85,B 0,C 180,E1 -5103.71,E2 -5103.71} C_VEL
LIN {X 0,Y 670.935,Z 325.573,A -85,B 0,C 180,E1 -5104.823,E2 -5104.823} C_VEL
LIN {X 0,Y 670.612,Z 351.086,A -85,B 0,C 180,E1 -5107.265,E2 -5107.265} C_VEL
LIN {X 0,Y 670.152,Z 380.644,A -85,B 0,C 180,E1 -5110.047,E2 -5110.047} C_VEL
LIN {X 0,Y 669.717,Z 407.033,A -85,B 0,C 180,E1 -5112.501,E2 -5112.501} C_VEL
LIN {X 0,Y 669.403,Z 435.673,A -85,B 0,C 180,E1 -5115.146,E2 -5115.146} C_VEL
LIN {X 0,Y 669.324,Z 441.34,A -85,B 0,C 180,E1 -5115.667,E2 -5115.667} C_VEL
LIN {X 0,Y 670.789,Z 456.46,A -85,B 0,C 180,E1 -5115.872,E2 -5115.872} C_VEL
LIN {X 0,Y 670.274,Z 580.33,A -85,B 0,C 180,E1 -5117.208,E2 -5117.208} C_VEL
LIN {X 0,Y 670.101,Z 594.431,A -85,B 0,C 180,E1 -5117.473,E2 -5117.473} C_VEL
LIN {X 0,Y 669.911,Z 608.171,A -85,B 0,C 180,E1 -5117.853,E2 -5117.853} C_VEL
LIN {X 0,Y 669.663,Z 620.651,A -85,B 0,C 180,E1 -5118.308,E2 -5118.308} C_VEL
LIN {X 0,Y 669.389,Z 633.722,A -85,B 0,C 180,E1 -5118.914,E2 -5118.914} C_VEL
LIN {X 0,Y 669.178,Z 645.605,A -85,B 0,C 180,E1 -5119.598,E2 -5119.598} C_VEL
LIN {X 0,Y 668.994,Z 656.491,A -85,B 0,C 180,E1 -5120.356,E2 -5120.356} C_VEL
LIN {X 0,Y 668.764,Z 667.291,A -85,B 0,C 180,E1 -5121.265,E2 -5121.265} C_VEL
LIN {X 0,Y 668.64,Z 676.214,A -85,B 0,C 180,E1 -5122.173,E2 -5122.173} C_VEL
LIN {X 0,Y 668.495,Z 684.789,A -85,B 0,C 180,E1 -5123.23,E2 -5123.23} C_VEL
LIN {X 0,Y 668.412,Z 691.712,A -85,B 0,C 180,E1 -5124.286,E2 -5124.286} C_VEL
LIN {X 0,Y 668.372,Z 697.881,A -85,B 0,C 180,E1 -5125.492,E2 -5125.492} C_VEL
LIN {X 0,Y 668.309,Z 701.434,A -85,B 0,C 180,E1 -5126.394,E2 -5126.394} C_VEL
LIN {X 0,Y 668.327,Z 704.91,A -85,B 0,C 180,E1 -5127.597,E2 -5127.597} C_VEL
LIN {X 0,Y 668.277,Z 706.91,A -85,B 0,C 180,E1 -5128.799,E2 -5128.799} C_VEL
LIN {X 0,Y 668.241,Z 707.604,A -85,B 0,C 180,E1 -5130,E2 -5130} C_VEL
LIN {X 0,Y 668.277,Z 706.918,A -85,B 0,C 180,E1 -5131.201,E2 -5131.201} C_VEL
LIN {X 0,Y 668.327,Z 704.899,A -85,B 0,C 180,E1 -5132.403,E2 -5132.403} C_VEL
LIN {X 0,Y 668.309,Z 701.466,A -85,B 0,C 180,E1 -5133.605,E2 -5133.605} C_VEL
LIN {X 0,Y 668.396,Z 696.495,A -85,B 0,C 180,E1 -5134.809,E2 -5134.809} C_VEL
LIN {X 0,Y 668.415,Z 691.737,A -85,B 0,C 180,E1 -5135.713,E2 -5135.713} C_VEL
LIN {X 0,Y 668.506,Z 683.655,A -85,B 0,C 180,E1 -5136.921,E2 -5136.921} C_VEL
LIN {X 0,Y 668.64,Z 676.217,A -85,B 0,C 180,E1 -5137.827,E2 -5137.827} C_VEL
LIN {X 0,Y 668.763,Z 667.311,A -85,B 0,C 180,E1 -5138.735,E2 -5138.735} C_VEL
LIN {X 0,Y 668.994,Z 656.525,A -85,B 0,C 180,E1 -5139.644,E2 -5139.644} C_VEL
LIN {X 0,Y 669.224,Z 644.814,A -85,B 0,C 180,E1 -5140.455,E2 -5140.455} C_VEL
LIN {X 0,Y 669.407,Z 632.325,A -85,B 0,C 180,E1 -5141.162,E2 -5141.162} C_VEL
LIN {X 0,Y 669.725,Z 618.834,A -85,B 0,C 180,E1 -5141.768,E2 -5141.768} C_VEL
LIN {X 0,Y 669.939,Z 605.812,A -85,B 0,C 180,E1 -5142.223,E2 -5142.223} C_VEL
LIN {X 0,Y 670.162,Z 591.871,A -85,B 0,C 180,E1 -5142.583,E2 -5142.583} C_VEL
LIN {X 0,Y 670.324,Z 577.422,A -85,B 0,C 180,E1 -5142.829,E2 -5142.829} C_VEL
LIN {X 0,Y 670.782,Z 454.419,A -85,B 0,C 180,E1 -5144.151,E2 -5144.151} C_VEL
LIN {X 0,Y 669.324,Z 441.397,A -85,B 0,C 180,E1 -5144.333,E2 -5144.333} C_VEL
LIN {X 0,Y 669.697,Z 410.482,A -85,B 0,C 180,E1 -5147.186,E2 -5147.186} C_VEL
LIN {X 0,Y 670.082,Z 384.128,A -85,B 0,C 180,E1 -5149.636,E2 -5149.636} C_VEL
LIN {X 0,Y 670.455,Z 359.547,A -85,B 0,C 180,E1 -5151.943,E2 -5151.943} C_VEL
LIN {X 0,Y 670.772,Z 337.462,A -85,B 0,C 180,E1 -5154.032,E2 -5154.032} C_VEL
LIN {X 0,Y 670.901,Z 325.443,A -85,B 0,C 180,E1 -5155.179,E2 -5155.179} C_VEL
LIN {X 0,Y 668.889,Z 314.725,A -85,B 0,C 180,E1 -5156.28,E2 -5156.28} C_VEL
LIN {X 0,Y 668.858,Z 314.724,A -85,B 0,C 180,E1 -5158.798,E2 -5158.798} C_VEL
LIN {X 0,Y 668.874,Z 314.721,A -85,B 0,C 180,E1 -5160.872,E2 -5160.872} C_VEL
LIN {X 0,Y 668.882,Z 314.723,A -85,B 0,C 180,E1 -5163.097,E2 -5163.097} C_VEL
LIN {X 0,Y 668.877,Z 314.722,A -85,B 0,C 180,E1 -5165.904,E2 -5165.904} C_VEL
LIN {X 0,Y 668.865,Z 314.721,A -85,B 0,C 180,E1 -5168.241,E2 -5168.241} C_VEL
LIN {X 0,Y 668.86,Z 314.722,A -85,B 0,C 180,E1 -5170.487,E2 -5170.487} C_VEL
LIN {X 0,Y 668.836,Z 314.731,A -85,B 0,C 180,E1 -5172.9,E2 -5172.9} C_VEL
LIN {X 0,Y 668.904,Z 314.722,A -85,B 0,C 180,E1 -5175.445,E2 -5175.445} C_VEL
LIN {X 0,Y 668.863,Z 314.722,A -85,B 0,C 180,E1 -5178.033,E2 -5178.033} C_VEL
LIN {X 0,Y 668.884,Z 314.726,A -85,B 0,C 180,E1 -5180.797,E2 -5180.797} C_VEL
LIN {X 0,Y 668.882,Z 314.723,A -85,B 0,C 180,E1 -5183.352,E2 -5183.352} C_VEL
LIN {X 0,Y 668.883,Z 314.72,A -85,B 0,C 180,E1 -5185.82,E2 -5185.82} C_VEL
LIN {X 0,Y 668.875,Z 314.73,A -85,B 0,C 180,E1 -5188.426,E2 -5188.426} C_VEL
LIN {X 0,Y 668.891,Z 314.726,A -85,B 0,C 180,E1 -5191.204,E2 -5191.204} C_VEL
LIN {X 0,Y 668.889,Z 314.725,A -85,B 0,C 180,E1 -5193.238,E2 -5193.238} C_VEL
LIN {X 0,Y 668.893,Z 314.751,A -85,B 0,C 180,E1 -5194.148,E2 -5194.148} C_VEL
LIN {X 0,Y 670.799,Z 325.053,A -85,B 0,C 180,E1 -5195.148,E2 -5195.148} C_VEL
LIN {X 0,Y 670.649,Z 350.037,A -85,B 0,C 180,E1 -5197.429,E2 -5197.429} C_VEL
LIN {X 0,Y 670.361,Z 377.079,A -85,B 0,C 180,E1 -5199.927,E2 -5199.927} C_VEL
LIN {X 0,Y 669.956,Z 406.694,A -85,B 0,C 180,E1 -5202.664,E2 -5202.664} C_VEL
LIN {X 0,Y 669.64,Z 431.622,A -85,B 0,C 180,E1 -5204.996,E2 -5204.996} C_VEL
LIN {X 0,Y 669.559,Z 439.51,A -85,B 0,C 180,E1 -5205.73,E2 -5205.73} C_VEL
LIN {X 0,Y 670.808,Z 450.568,A -85,B 0,C 180,E1 -5205.892,E2 -5205.892} C_VEL
LIN {X 0,Y 670.268,Z 578.398,A -85,B 0,C 180,E1 -5207.323,E2 -5207.323} C_VEL
LIN {X 0,Y 670.068,Z 592.279,A -85,B 0,C 180,E1 -5207.588,E2 -5207.588} C_VEL
LIN {X 0,Y 669.896,Z 605.983,A -85,B 0,C 180,E1 -5207.968,E2 -5207.968} C_VEL
LIN {X 0,Y 669.651,Z 619.281,A -85,B 0,C 180,E1 -5208.461,E2 -5208.461} C_VEL
LIN {X 0,Y 669.388,Z 631.997,A -85,B 0,C 180,E1 -5209.067,E2 -5209.067} C_VEL
LIN {X 0,Y 669.226,Z 643.627,A -85,B 0,C 180,E1 -5209.751,E2 -5209.751} C_VEL
LIN {X 0,Y 669.041,Z 654.278,A -85,B 0,C 180,E1 -5210.509,E2 -5210.509} C_VEL
LIN {X 0,Y 668.806,Z 664.799,A -85,B 0,C 180,E1 -5211.417,E2 -5211.417} C_VEL
LIN {X 0,Y 668.634,Z 673.46,A -85,B 0,C 180,E1 -5212.324,E2 -5212.324} C_VEL
LIN {X 0,Y 668.508,Z 680.665,A -85,B 0,C 180,E1 -5213.231,E2 -5213.231} C_VEL
LIN {X 0,Y 668.389,Z 687.6,A -85,B 0,C 180,E1 -5214.287,E2 -5214.287} C_VEL
LIN {X 0,Y 668.359,Z 693.781,A -85,B 0,C 180,E1 -5215.492,E2 -5215.492} C_VEL
LIN {X 0,Y 668.278,Z 697.332,A -85,B 0,C 180,E1 -5216.395,E2 -5216.395} C_VEL
LIN {X 0,Y 668.297,Z 700.736,A -85,B 0,C 180,E1 -5217.597,E2 -5217.597} C_VEL
LIN {X 0,Y 668.241,Z 702.794,A -85,B 0,C 180,E1 -5218.799,E2 -5218.799} C_VEL
LIN {X 0,Y 668.222,Z 703.517,A -85,B 0,C 180,E1 -5220,E2 -5220} C_VEL
LIN {X 0,Y 668.239,Z 702.879,A -85,B 0,C 180,E1 -5221.201,E2 -5221.201} C_VEL
LIN {X 0,Y 668.296,Z 700.938,A -85,B 0,C 180,E1 -5222.403,E2 -5222.403} C_VEL
LIN {X 0,Y 668.278,Z 697.619,A -85,B 0,C 180,E1 -5223.606,E2 -5223.606} C_VEL
LIN {X 0,Y 668.386,Z 692.825,A -85,B 0,C 180,E1 -5224.809,E2 -5224.809} C_VEL
LIN {X 0,Y 668.39,Z 687.117,A -85,B 0,C 180,E1 -5225.883,E2 -5225.883} C_VEL
LIN {X 0,Y 668.506,Z 681.333,A -85,B 0,C 180,E1 -5226.77,E2 -5226.77} C_VEL
LIN {X 0,Y 668.608,Z 674.251,A -85,B 0,C 180,E1 -5227.676,E2 -5227.676} C_VEL
LIN {X 0,Y 668.789,Z 665.76,A -85,B 0,C 180,E1 -5228.583,E2 -5228.583} C_VEL
LIN {X 0,Y 669.017,Z 655.492,A -85,B 0,C 180,E1 -5229.492,E2 -5229.492} C_VEL
LIN {X 0,Y 669.198,Z 644.392,A -85,B 0,C 180,E1 -5230.298,E2 -5230.298} C_VEL
LIN {X 0,Y 669.417,Z 632.404,A -85,B 0,C 180,E1 -5231.009,E2 -5231.009} C_VEL
LIN {X 0,Y 669.656,Z 621.514,A -85,B 0,C 180,E1 -5231.54,E2 -5231.54} C_VEL
LIN {X 0,Y 669.913,Z 607.943,A -85,B 0,C 180,E1 -5232.071,E2 -5232.071} C_VEL
LIN {X 0,Y 670.059,Z 593.411,A -85,B 0,C 180,E1 -5232.489,E2 -5232.489} C_VEL
LIN {X 0,Y 670.244,Z 580.141,A -85,B 0,C 180,E1 -5232.754,E2 -5232.754} C_VEL
LIN {X 0,Y 670.393,Z 549.475,A -85,B 0,C 180,E1 -5233.116,E2 -5233.116} C_VEL
LIN {X 0,Y 670.725,Z 448.438,A -85,B 0,C 180,E1 -5234.226,E2 -5234.226} C_VEL
LIN {X 0,Y 669.523,Z 439.53,A -85,B 0,C 180,E1 -5234.368,E2 -5234.368} C_VEL
LIN {X 0,Y 669.904,Z 416.372,A -85,B 0,C 180,E1 -5236.554,E2 -5236.554} C_VEL
LIN {X 0,Y 670.371,Z 388.29,A -85,B 0,C 180,E1 -5239.216,E2 -5239.216} C_VEL
LIN {X 0,Y 670.835,Z 359.649,A -85,B 0,C 180,E1 -5241.937,E2 -5241.937} C_VEL
LIN {X 0,Y 671.064,Z 345.871,A -85,B 0,C 180,E1 -5243.252,E2 -5243.252} C_VEL
LIN {X 0,Y 670.565,Z 342.083,A -85,B 0,C 180,E1 -5243.634,E2 -5243.634} C_VEL
LIN {X 0,Y 668.178,Z 336.215,A -85,B 0,C 180,E1 -5244.28,E2 -5244.28} C_VEL
LIN {X 0,Y 665.893,Z 331.566,A -85,B 0,C 180,E1 -5244.803,E2 -5244.803} C_VEL
LIN {X 0,Y 664.283,Z 326.695,A -85,B 0,C 180,E1 -5245.328,E2 -5245.328} C_VEL
LIN {X 0,Y 661.864,Z 315.599,A -85,B 0,C 180,E1 -5246.517,E2 -5246.517} C_VEL
LIN {X 0,Y 661.886,Z 315.598,A -85,B 0,C 180,E1 -5249.131,E2 -5249.131} C_VEL
LIN {X 0,Y 661.857,Z 315.603,A -85,B 0,C 180,E1 -5251.237,E2 -5251.237} C_VEL
LIN {X 0,Y 661.877,Z 315.59,A -85,B 0,C 180,E1 -5254.117,E2 -5254.117} C_VEL
